LIN {X 0,Y 417.508,Z 538.945,A -85,B 0,C 180,E1 -10179.202,E2 -10179.202} C_VEL
LIN {X 0,Y 417.931,Z 531.783,A -85,B 0,C 180,E1 -10180.905,E2 -10180.905} C_VEL
LIN {X 0,Y 418.426,Z 524.272,A -85,B 0,C 180,E1 -10182.366,E2 -10182.366} C_VEL
LIN {X 0,Y 419.126,Z 515.227,A -85,B 0,C 180,E1 -10183.824,E2 -10183.824} C_VEL
LIN {X 0,Y 419.941,Z 504.249,A -85,B 0,C 180,E1 -10185.283,E2 -10185.283} C_VEL
LIN {X 0,Y 420.839,Z 493.102,A -85,B 0,C 180,E1 -10186.493,E2 -10186.493} C_VEL
LIN {X 0,Y 421.825,Z 480.792,A -85,B 0,C 180,E1 -10187.576,E2 -10187.576} C_VEL
LIN {X 0,Y 422.664,Z 467.695,A -85,B 0,C 180,E1 -10188.494,E2 -10188.494} C_VEL
LIN {X 0,Y 423.488,Z 453.313,A -85,B 0,C 180,E1 -10189.262,E2 -10189.262} C_VEL
LIN {X 0,Y 424.154,Z 439.428,A -85,B 0,C 180,E1 -10189.794,E2 -10189.794} C_VEL
LIN {X 0,Y 424.598,Z 424.854,A -85,B 0,C 180,E1 -10190.15,E2 -10190.15} C_VEL
LIN {X 0,Y 426.165,Z 318.753,A -85,B 0,C 180,E1 -10192.051,E2 -10192.051} C_VEL
LIN {X 0,Y 422.715,Z 297.962,A -85,B 0,C 180,E1 -10192.643,E2 -10192.643} C_VEL
LIN {X 0,Y 424.107,Z 281.691,A -85,B 0,C 180,E1 -10195.259,E2 -10195.259} C_VEL
LIN {X 0,Y 423.846,Z 278.694,A -85,B 0,C 180,E1 -10195.785,E2 -10195.785} C_VEL
LIN {X 0,Y 420.942,Z 266.303,A -85,B 0,C 180,E1 -10198.141,E2 -10198.141} C_VEL
LIN {X 0,Y 418.292,Z 256.11,A -85,B 0,C 180,E1 -10200.218,E2 -10200.218} C_VEL
LIN {X 0,Y 418.246,Z 256.011,A -85,B 0,C 180,E1 -10203.677,E2 -10203.677} C_VEL
LIN {X 0,Y 418.237,Z 255.991,A -85,B 0,C 180,E1 -10207.224,E2 -10207.224} C_VEL
LIN {X 0,Y 418.246,Z 256.012,A -85,B 0,C 180,E1 -10209.682,E2 -10209.682} C_VEL
LIN {X 0,Y 418.281,Z 256.01,A -85,B 0,C 180,E1 -10212.329,E2 -10212.329} C_VEL
LIN {X 0,Y 418.248,Z 256.006,A -85,B 0,C 180,E1 -10215.11,E2 -10215.11} C_VEL
LIN {X 0,Y 418.236,Z 256.008,A -85,B 0,C 180,E1 -10217.767,E2 -10217.767} C_VEL
LIN {X 0,Y 418.255,Z 256.011,A -85,B 0,C 180,E1 -10220.618,E2 -10220.618} C_VEL
LIN {X 0,Y 418.241,Z 255.998,A -85,B 0,C 180,E1 -10223.976,E2 -10223.976} C_VEL
LIN {X 0,Y 418.253,Z 256.009,A -85,B 0,C 180,E1 -10227.156,E2 -10227.156} C_VEL
LIN {X 0,Y 418.269,Z 255.993,A -85,B 0,C 180,E1 -10230.839,E2 -10230.839} C_VEL
LIN {X 0,Y 418.265,Z 256.01,A -85,B 0,C 180,E1 -10234.096,E2 -10234.096} C_VEL
LIN {X 0,Y 418.232,Z 256.011,A -85,B 0,C 180,E1 -10237.264,E2 -10237.264} C_VEL
LIN {X 0,Y 418.277,Z 256.006,A -85,B 0,C 180,E1 -10240.364,E2 -10240.364} C_VEL
LIN {X 0,Y 418.311,Z 256,A -85,B 0,C 180,E1 -10243.405,E2 -10243.405} C_VEL
LIN {X 0,Y 418.34,Z 255.996,A -85,B 0,C 180,E1 -10246.999,E2 -10246.999} C_VEL
LIN {X 0,Y 418.335,Z 255.998,A -85,B 0,C 180,E1 -10250.329,E2 -10250.329} C_VEL
LIN {X 0,Y 418.486,Z 255.973,A -85,B 0,C 180,E1 -10253.249,E2 -10253.249} C_VEL
LIN {X 0,Y 418.335,Z 256,A -85,B 0,C 180,E1 -10255.182,E2 -10255.182} C_VEL
LIN {X 0,Y 418.539,Z 255.971,A -85,B 0,C 180,E1 -10258.076,E2 -10258.076} C_VEL
LIN {X 0,Y 418.666,Z 255.958,A -85,B 0,C 180,E1 -10260,E2 -10260} C_VEL
LIN {X 0,Y 418.505,Z 255.971,A -85,B 0,C 180,E1 -10262.888,E2 -10262.888} C_VEL
LIN {X 0,Y 418.488,Z 255.974,A -85,B 0,C 180,E1 -10266.751,E2 -10266.751} C_VEL
LIN {X 0,Y 418.394,Z 255.989,A -85,B 0,C 180,E1 -10268.696,E2 -10268.696} C_VEL
LIN {X 0,Y 418.31,Z 255.998,A -85,B 0,C 180,E1 -10271.632,E2 -10271.632} C_VEL
LIN {X 0,Y 418.298,Z 256.002,A -85,B 0,C 180,E1 -10274.598,E2 -10274.598} C_VEL
LIN {X 0,Y 418.283,Z 256.007,A -85,B 0,C 180,E1 -10277.604,E2 -10277.604} C_VEL
LIN {X 0,Y 418.245,Z 256.005,A -85,B 0,C 180,E1 -10280.664,E2 -10280.664} C_VEL
LIN {X 0,Y 418.284,Z 256.002,A -85,B 0,C 180,E1 -10283.782,E2 -10283.782} C_VEL
LIN {X 0,Y 418.307,Z 255.999,A -85,B 0,C 180,E1 -10287.071,E2 -10287.071} C_VEL
LIN {X 0,Y 418.241,Z 256.001,A -85,B 0,C 180,E1 -10290.273,E2 -10290.273} C_VEL
LIN {X 0,Y 418.246,Z 256.004,A -85,B 0,C 180,E1 -10293.678,E2 -10293.678} C_VEL
LIN {X 0,Y 418.243,Z 256.014,A -85,B 0,C 180,E1 -10297.224,E2 -10297.224} C_VEL
LIN {X 0,Y 418.246,Z 255.998,A -85,B 0,C 180,E1 -10299.683,E2 -10299.683} C_VEL
LIN {X 0,Y 418.228,Z 256.014,A -85,B 0,C 180,E1 -10302.322,E2 -10302.322} C_VEL
LIN {X 0,Y 418.239,Z 256.011,A -85,B 0,C 180,E1 -10305.11,E2 -10305.11} C_VEL
LIN {X 0,Y 418.242,Z 256.004,A -85,B 0,C 180,E1 -10307.768,E2 -10307.768} C_VEL
LIN {X 0,Y 418.259,Z 255.993,A -85,B 0,C 180,E1 -10310.619,E2 -10310.619} C_VEL
LIN {X 0,Y 418.243,Z 256.013,A -85,B 0,C 180,E1 -10313.977,E2 -10313.977} C_VEL
LIN {X 0,Y 418.255,Z 256.107,A -85,B 0,C 180,E1 -10317.276,E2 -10317.276} C_VEL
LIN {X 0,Y 421.436,Z 269.127,A -85,B 0,C 180,E1 -10320.132,E2 -10320.132} C_VEL
LIN {X 0,Y 423.369,Z 278.645,A -85,B 0,C 180,E1 -10322.1,E2 -10322.1} C_VEL
LIN {X 0,Y 422.447,Z 290.987,A -85,B 0,C 180,E1 -10324.371,E2 -10324.371} C_VEL
LIN {X 0,Y 421.363,Z 305.324,A -85,B 0,C 180,E1 -10326.963,E2 -10326.963} C_VEL
LIN {X 0,Y 420.9,Z 313.173,A -85,B 0,C 180,E1 -10328.32,E2 -10328.32} C_VEL
LIN {X 0,Y 425.453,Z 338.255,A -85,B 0,C 180,E1 -10329.003,E2 -10329.003} C_VEL
LIN {X 0,Y 424.456,Z 426.611,A -85,B 0,C 180,E1 -10330.441,E2 -10330.441} C_VEL
LIN {X 0,Y 423.954,Z 439.651,A -85,B 0,C 180,E1 -10330.843,E2 -10330.843} C_VEL
LIN {X 0,Y 423.469,Z 452.234,A -85,B 0,C 180,E1 -10331.433,E2 -10331.433} C_VEL
LIN {X 0,Y 422.684,Z 464.51,A -85,B 0,C 180,E1 -10332.211,E2 -10332.211} C_VEL
LIN {X 0,Y 421.704,Z 476.092,A -85,B 0,C 180,E1 -10333.168,E2 -10333.168} C_VEL
LIN {X 0,Y 420.799,Z 486.5,A -85,B 0,C 180,E1 -10334.253,E2 -10334.253} C_VEL
LIN {X 0,Y 419.845,Z 496.326,A -85,B 0,C 180,E1 -10335.523,E2 -10335.523} C_VEL
LIN {X 0,Y 419.149,Z 503.803,A -85,B 0,C 180,E1 -10336.704,E2 -10336.704} C_VEL
LIN {X 0,Y 418.6,Z 511.176,A -85,B 0,C 180,E1 -10338.132,E2 -10338.132} C_VEL
LIN {X 0,Y 418.229,Z 514.558,A -85,B 0,C 180,E1 -10338.9,E2 -10338.9} C_VEL
LIN {X 0,Y 417.29,Z 517.409,A -85,B 0,C 180,E1 -10339.603,E2 -10339.603} C_VEL
LIN {X 0,Y 414.133,Z 521.613,A -85,B 0,C 180,E1 -10340.763,E2 -10340.763} C_VEL
LIN {X 0,Y 411.055,Z 525.123,A -85,B 0,C 180,E1 -10341.978,E2 -10341.978} C_VEL
LIN {X 0,Y 410.253,Z 526.877,A -85,B 0,C 180,E1 -10342.756,E2 -10342.756} C_VEL
LIN {X 0,Y 410.07,Z 529.255,A -85,B 0,C 180,E1 -10344.098,E2 -10344.098} C_VEL
LIN {X 0,Y 410.043,Z 530.517,A -85,B 0,C 180,E1 -10345.084,E2 -10345.084} C_VEL
LIN {X 0,Y 409.969,Z 531.939,A -85,B 0,C 180,E1 -10347.052,E2 -10347.052} C_VEL
LIN {X 0,Y 410.003,Z 532.078,A -85,B 0,C 180,E1 -10348.035,E2 -10348.035} C_VEL
LIN {X 0,Y 409.931,Z 531.25,A -85,B 0,C 180,E1 -10350,E2 -10350} C_VEL
LIN {X 0,Y 410.075,Z 528.965,A -85,B 0,C 180,E1 -10351.964,E2 -10351.964} C_VEL
LIN {X 0,Y 410.324,Z 526.18,A -85,B 0,C 180,E1 -10353.437,E2 -10353.437} C_VEL
LIN {X 0,Y 410.454,Z 522.443,A -85,B 0,C 180,E1 -10354.911,E2 -10354.911} C_VEL
LIN {X 0,Y 410.864,Z 517.636,A -85,B 0,C 180,E1 -10356.383,E2 -10356.383} C_VEL
LIN {X 0,Y 411.338,Z 511.624,A -85,B 0,C 180,E1 -10357.856,E2 -10357.856} C_VEL
LIN {X 0,Y 411.984,Z 504.185,A -85,B 0,C 180,E1 -10359.326,E2 -10359.326} C_VEL
LIN {X 0,Y 412.859,Z 494.877,A -85,B 0,C 180,E1 -10360.792,E2 -10360.792} C_VEL
LIN {X 0,Y 413.798,Z 484.254,A -85,B 0,C 180,E1 -10362.133,E2 -10362.133} C_VEL
LIN {X 0,Y 414.707,Z 473.337,A -85,B 0,C 180,E1 -10363.225,E2 -10363.225} C_VEL
LIN {X 0,Y 415.303,Z 464.403,A -85,B 0,C 180,E1 -10363.954,E2 -10363.954} C_VEL
LIN {X 0,Y 416.025,Z 453.249,A -85,B 0,C 180,E1 -10364.678,E2 -10364.678} C_VEL
LIN {X 0,Y 416.72,Z 440.712,A -85,B 0,C 180,E1 -10365.278,E2 -10365.278} C_VEL
LIN {X 0,Y 417.121,Z 427.911,A -85,B 0,C 180,E1 -10365.697,E2 -10365.697} C_VEL
LIN {X 0,Y 417.48,Z 404.6,A -85,B 0,C 180,E1 -10366.111,E2 -10366.111} C_VEL
LIN {X 0,Y 418.004,Z 337.982,A -85,B 0,C 180,E1 -10367.196,E2 -10367.196} C_VEL
LIN {X 0,Y 413.749,Z 313.265,A -85,B 0,C 180,E1 -10367.842,E2 -10367.842} C_VEL
LIN {X 0,Y 413.723,Z 312.244,A -85,B 0,C 180,E1 -10367.956,E2 -10367.956} C_VEL
LIN {X 0,Y 415.029,Z 293.533,A -85,B 0,C 180,E1 -10371.351,E2 -10371.351} C_VEL
LIN {X 0,Y 416.17,Z 279.659,A -85,B 0,C 180,E1 -10373.909,E2 -10373.909} C_VEL
LIN {X 0,Y 413.971,Z 268.598,A -85,B 0,C 180,E1 -10376.193,E2 -10376.193} C_VEL
LIN {X 0,Y 411.272,Z 256.972,A -85,B 0,C 180,E1 -10378.736,E2 -10378.736} C_VEL
LIN {X 0,Y 411.168,Z 256.892,A -85,B 0,C 180,E1 -10381.996,E2 -10381.996} C_VEL
LIN {X 0,Y 411.212,Z 256.877,A -85,B 0,C 180,E1 -10384.878,E2 -10384.878} C_VEL
LIN {X 0,Y 411.206,Z 256.884,A -85,B 0,C 180,E1 -10388.168,E2 -10388.168} C_VEL
LIN {X 0,Y 411.164,Z 256.887,A -85,B 0,C 180,E1 -10391.228,E2 -10391.228} C_VEL
LIN {X 0,Y 411.179,Z 256.886,A -85,B 0,C 180,E1 -10394.489,E2 -10394.489} C_VEL
LIN {X 0,Y 411.175,Z 256.889,A -85,B 0,C 180,E1 -10398.194,E2 -10398.194} C_VEL
LIN {X 0,Y 411.21,Z 256.873,A -85,B 0,C 180,E1 -10400.774,E2 -10400.774} C_VEL
LIN {X 0,Y 411.197,Z 256.887,A -85,B 0,C 180,E1 -10404.471,E2 -10404.471} C_VEL
LIN {X 0,Y 411.204,Z 256.87,A -85,B 0,C 180,E1 -10406.872,E2 -10406.872} C_VEL
LIN {X 0,Y 411.237,Z 256.886,A -85,B 0,C 180,E1 -10410.641,E2 -10410.641} C_VEL
LIN {X 0,Y 411.234,Z 256.883,A -85,B 0,C 180,E1 -10413.618,E2 -10413.618} C_VEL
LIN {X 0,Y 411.192,Z 256.888,A -85,B 0,C 180,E1 -10416.851,E2 -10416.851} C_VEL
LIN {X 0,Y 411.209,Z 256.881,A -85,B 0,C 180,E1 -10420.05,E2 -10420.05} C_VEL
LIN {X 0,Y 411.258,Z 256.88,A -85,B 0,C 180,E1 -10423.13,E2 -10423.13} C_VEL
LIN {X 0,Y 411.3,Z 256.879,A -85,B 0,C 180,E1 -10426.895,E2 -10426.895} C_VEL
LIN {X 0,Y 411.287,Z 256.871,A -85,B 0,C 180,E1 -10430.161,E2 -10430.161} C_VEL
LIN {X 0,Y 411.45,Z 256.856,A -85,B 0,C 180,E1 -10433.132,E2 -10433.132} C_VEL
LIN {X 0,Y 411.305,Z 256.866,A -85,B 0,C 180,E1 -10435.099,E2 -10435.099} C_VEL
LIN {X 0,Y 411.507,Z 256.85,A -85,B 0,C 180,E1 -10438.042,E2 -10438.042} C_VEL
LIN {X 0,Y 411.635,Z 256.831,A -85,B 0,C 180,E1 -10440,E2 -10440} C_VEL
LIN {X 0,Y 411.459,Z 256.856,A -85,B 0,C 180,E1 -10442.937,E2 -10442.937} C_VEL
LIN {X 0,Y 411.453,Z 256.854,A -85,B 0,C 180,E1 -10446.867,E2 -10446.867} C_VEL
LIN {X 0,Y 411.347,Z 256.869,A -85,B 0,C 180,E1 -10448.845,E2 -10448.845} C_VEL
LIN {X 0,Y 411.277,Z 256.872,A -85,B 0,C 180,E1 -10451.833,E2 -10451.833} C_VEL
LIN {X 0,Y 411.253,Z 256.877,A -85,B 0,C 180,E1 -10454.853,E2 -10454.853} C_VEL
LIN {X 0,Y 411.246,Z 256.883,A -85,B 0,C 180,E1 -10457.915,E2 -10457.915} C_VEL
LIN {X 0,Y 411.19,Z 256.884,A -85,B 0,C 180,E1 -10461.034,E2 -10461.034} C_VEL
LIN {X 0,Y 411.22,Z 256.883,A -85,B 0,C 180,E1 -10464.216,E2 -10464.216} C_VEL
LIN {X 0,Y 411.254,Z 256.882,A -85,B 0,C 180,E1 -10467.478,E2 -10467.478} C_VEL
LIN {X 0,Y 411.192,Z 256.872,A -85,B 0,C 180,E1 -10470.847,E2 -10470.847} C_VEL
LIN {X 0,Y 411.201,Z 256.888,A -85,B 0,C 180,E1 -10474.334,E2 -10474.334} C_VEL
LIN {X 0,Y 411.196,Z 256.881,A -85,B 0,C 180,E1 -10477.973,E2 -10477.973} C_VEL
LIN {X 0,Y 411.178,Z 256.889,A -85,B 0,C 180,E1 -10480.504,E2 -10480.504} C_VEL
LIN {X 0,Y 411.169,Z 256.886,A -85,B 0,C 180,E1 -10483.134,E2 -10483.134} C_VEL
LIN {X 0,Y 411.164,Z 256.883,A -85,B 0,C 180,E1 -10485.881,E2 -10485.881} C_VEL
LIN {X 0,Y 411.16,Z 256.86,A -85,B 0,C 180,E1 -10488.772,E2 -10488.772} C_VEL
LIN {X 0,Y 411.203,Z 256.888,A -85,B 0,C 180,E1 -10491.832,E2 -10491.832} C_VEL
LIN {X 0,Y 411.208,Z 256.871,A -85,B 0,C 180,E1 -10495.122,E2 -10495.122} C_VEL
LIN {X 0,Y 411.163,Z 256.876,A -85,B 0,C 180,E1 -10498.003,E2 -10498.003} C_VEL
LIN {X 0,Y 411.24,Z 257.068,A -85,B 0,C 180,E1 -10499.867,E2 -10499.867} C_VEL
LIN {X 0,Y 414.703,Z 270.774,A -85,B 0,C 180,E1 -10502.581,E2 -10502.581} C_VEL
LIN {X 0,Y 416.945,Z 281.265,A -85,B 0,C 180,E1 -10504.544,E2 -10504.544} C_VEL
LIN {X 0,Y 415.497,Z 297.774,A -85,B 0,C 180,E1 -10507.248,E2 -10507.248} C_VEL
LIN {X 0,Y 418.94,Z 319.913,A -85,B 0,C 180,E1 -10507.874,E2 -10507.874} C_VEL
LIN {X 0,Y 417.188,Z 430.973,A -85,B 0,C 180,E1 -10509.894,E2 -10509.894} C_VEL
LIN {X 0,Y 416.62,Z 445.021,A -85,B 0,C 180,E1 -10510.318,E2 -10510.318} C_VEL
LIN {X 0,Y 415.957,Z 458.882,A -85,B 0,C 180,E1 -10510.942,E2 -10510.942} C_VEL
LIN {X 0,Y 415.259,Z 471.531,A -85,B 0,C 180,E1 -10511.701,E2 -10511.701} C_VEL
LIN {X 0,Y 414.285,Z 484.97,A -85,B 0,C 180,E1 -10512.73,E2 -10512.73} C_VEL
LIN {X 0,Y 413.404,Z 496.539,A -85,B 0,C 180,E1 -10513.837,E2 -10513.837} C_VEL
LIN {X 0,Y 412.579,Z 506.143,A -85,B 0,C 180,E1 -10514.944,E2 -10514.944} C_VEL
LIN {X 0,Y 411.84,Z 516.768,A -85,B 0,C 180,E1 -10516.42,E2 -10516.42} C_VEL
LIN {X 0,Y 411.257,Z 525.627,A -85,B 0,C 180,E1 -10517.917,E2 -10517.917} C_VEL
LIN {X 0,Y 410.611,Z 533.98,A -85,B 0,C 180,E1 -10519.647,E2 -10519.647} C_VEL
LIN {X 0,Y 410.328,Z 539.839,A -85,B 0,C 180,E1 -10521.133,E2 -10521.133} C_VEL
LIN {X 0,Y 410.152,Z 544.584,A -85,B 0,C 180,E1 -10522.617,E2 -10522.617} C_VEL
LIN {X 0,Y 409.985,Z 548.373,A -85,B 0,C 180,E1 -10524.097,E2 -10524.097} C_VEL
LIN {X 0,Y 409.976,Z 550.404,A -85,B 0,C 180,E1 -10525.083,E2 -10525.083} C_VEL
LIN {X 0,Y 409.921,Z 553.34,A -85,B 0,C 180,E1 -10527.052,E2 -10527.052} C_VEL
LIN {X 0,Y 409.964,Z 554.267,A -85,B 0,C 180,E1 -10528.035,E2 -10528.035} C_VEL
LIN {X 0,Y 409.924,Z 555.055,A -85,B 0,C 180,E1 -10530,E2 -10530} C_VEL
LIN {X 0,Y 409.964,Z 554.426,A -85,B 0,C 180,E1 -10531.965,E2 -10531.965} C_VEL
LIN {X 0,Y 409.918,Z 552.354,A -85,B 0,C 180,E1 -10533.932,E2 -10533.932} C_VEL
LIN {X 0,Y 410.004,Z 548.817,A -85,B 0,C 180,E1 -10535.903,E2 -10535.903} C_VEL
LIN {X 0,Y 410.185,Z 543.719,A -85,B 0,C 180,E1 -10537.878,E2 -10537.878} C_VEL
LIN {X 0,Y 410.474,Z 538.77,A -85,B 0,C 180,E1 -10539.361,E2 -10539.361} C_VEL
LIN {X 0,Y 410.926,Z 531.608,A -85,B 0,C 180,E1 -10541.093,E2 -10541.093} C_VEL
LIN {X 0,Y 411.588,Z 522.719,A -85,B 0,C 180,E1 -10542.825,E2 -10542.825} C_VEL
LIN {X 0,Y 412.298,Z 513.396,A -85,B 0,C 180,E1 -10544.31,E2 -10544.31} C_VEL
LIN {X 0,Y 413.146,Z 503.071,A -85,B 0,C 180,E1 -10545.667,E2 -10545.667} C_VEL
LIN {X 0,Y 414.147,Z 491.652,A -85,B 0,C 180,E1 -10546.894,E2 -10546.894} C_VEL
LIN {X 0,Y 415.173,Z 478.997,A -85,B 0,C 180,E1 -10547.995,E2 -10547.995} C_VEL
LIN {X 0,Y 415.992,Z 466.908,A -85,B 0,C 180,E1 -10548.838,E2 -10548.838} C_VEL
LIN {X 0,Y 416.76,Z 453.384,A -85,B 0,C 180,E1 -10549.569,E2 -10549.569} C_VEL
LIN {X 0,Y 417.464,Z 439.087,A -85,B 0,C 180,E1 -10550.124,E2 -10550.124} C_VEL
LIN {X 0,Y 417.928,Z 424.273,A -85,B 0,C 180,E1 -10550.486,E2 -10550.486} C_VEL
LIN {X 0,Y 419.563,Z 319.793,A -85,B 0,C 180,E1 -10552.386,E2 -10552.386} C_VEL
LIN {X 0,Y 415.969,Z 297.92,A -85,B 0,C 180,E1 -10553.031,E2 -10553.031} C_VEL
LIN {X 0,Y 417.324,Z 283.314,A -85,B 0,C 180,E1 -10555.431,E2 -10555.431} C_VEL
LIN {X 0,Y 416.994,Z 280.233,A -85,B 0,C 180,E1 -10555.989,E2 -10555.989} C_VEL
LIN {X 0,Y 414.402,Z 269.167,A -85,B 0,C 180,E1 -10558.129,E2 -10558.129} C_VEL
LIN {X 0,Y 411.232,Z 256.989,A -85,B 0,C 180,E1 -10560.647,E2 -10560.647} C_VEL
LIN {X 0,Y 411.204,Z 256.889,A -85,B 0,C 180,E1 -10564.333,E2 -10564.333} C_VEL
LIN {X 0,Y 411.191,Z 256.879,A -85,B 0,C 180,E1 -10567.973,E2 -10567.973} C_VEL
LIN {X 0,Y 411.202,Z 256.883,A -85,B 0,C 180,E1 -10571.235,E2 -10571.235} C_VEL
LIN {X 0,Y 411.224,Z 256.877,A -85,B 0,C 180,E1 -10574.483,E2 -10574.483} C_VEL
LIN {X 0,Y 411.174,Z 256.882,A -85,B 0,C 180,E1 -10578.194,E2 -10578.194} C_VEL
LIN {X 0,Y 411.219,Z 256.887,A -85,B 0,C 180,E1 -10580.776,E2 -10580.776} C_VEL
LIN {X 0,Y 411.195,Z 256.876,A -85,B 0,C 180,E1 -10584.471,E2 -10584.471} C_VEL
LIN {X 0,Y 411.202,Z 256.887,A -85,B 0,C 180,E1 -10586.873,E2 -10586.873} C_VEL
LIN {X 0,Y 411.235,Z 256.866,A -85,B 0,C 180,E1 -10590.642,E2 -10590.642} C_VEL
LIN {X 0,Y 411.232,Z 256.885,A -85,B 0,C 180,E1 -10593.619,E2 -10593.619} C_VEL
LIN {X 0,Y 411.197,Z 256.887,A -85,B 0,C 180,E1 -10596.852,E2 -10596.852} C_VEL
LIN {X 0,Y 411.209,Z 256.885,A -85,B 0,C 180,E1 -10600.05,E2 -10600.05} C_VEL
LIN {X 0,Y 411.257,Z 256.878,A -85,B 0,C 180,E1 -10603.131,E2 -10603.131} C_VEL
LIN {X 0,Y 411.299,Z 256.873,A -85,B 0,C 180,E1 -10606.896,E2 -10606.896} C_VEL
LIN {X 0,Y 411.287,Z 256.877,A -85,B 0,C 180,E1 -10610.161,E2 -10610.161} C_VEL
LIN {X 0,Y 411.45,Z 256.849,A -85,B 0,C 180,E1 -10613.133,E2 -10613.133} C_VEL
LIN {X 0,Y 411.306,Z 256.875,A -85,B 0,C 180,E1 -10615.099,E2 -10615.099} C_VEL
LIN {X 0,Y 411.508,Z 256.847,A -85,B 0,C 180,E1 -10618.043,E2 -10618.043} C_VEL
LIN {X 0,Y 411.636,Z 256.834,A -85,B 0,C 180,E1 -10620,E2 -10620} C_VEL
LIN {X 0,Y 411.46,Z 256.848,A -85,B 0,C 180,E1 -10622.938,E2 -10622.938} C_VEL
LIN {X 0,Y 411.455,Z 256.851,A -85,B 0,C 180,E1 -10626.867,E2 -10626.867} C_VEL
LIN {X 0,Y 411.349,Z 256.868,A -85,B 0,C 180,E1 -10628.846,E2 -10628.846} C_VEL
LIN {X 0,Y 411.278,Z 256.875,A -85,B 0,C 180,E1 -10631.833,E2 -10631.833} C_VEL
LIN {X 0,Y 411.255,Z 256.881,A -85,B 0,C 180,E1 -10634.853,E2 -10634.853} C_VEL
LIN {X 0,Y 411.248,Z 256.881,A -85,B 0,C 180,E1 -10637.916,E2 -10637.916} C_VEL
LIN {X 0,Y 411.192,Z 256.887,A -85,B 0,C 180,E1 -10641.035,E2 -10641.035} C_VEL
LIN {X 0,Y 411.223,Z 256.88,A -85,B 0,C 180,E1 -10644.216,E2 -10644.216} C_VEL
LIN {X 0,Y 411.255,Z 256.872,A -85,B 0,C 180,E1 -10647.478,E2 -10647.478} C_VEL
LIN {X 0,Y 411.186,Z 256.884,A -85,B 0,C 180,E1 -10650.848,E2 -10650.848} C_VEL
LIN {X 0,Y 411.204,Z 256.879,A -85,B 0,C 180,E1 -10654.334,E2 -10654.334} C_VEL
LIN {X 0,Y 411.196,Z 256.888,A -85,B 0,C 180,E1 -10657.974,E2 -10657.974} C_VEL
LIN {X 0,Y 411.162,Z 256.891,A -85,B 0,C 180,E1 -10661.229,E2 -10661.229} C_VEL
LIN {X 0,Y 411.176,Z 256.883,A -85,B 0,C 180,E1 -10664.491,E2 -10664.491} C_VEL
LIN {X 0,Y 411.179,Z 256.885,A -85,B 0,C 180,E1 -10668.196,E2 -10668.196} C_VEL
LIN {X 0,Y 411.223,Z 256.866,A -85,B 0,C 180,E1 -10670.777,E2 -10670.777} C_VEL
LIN {X 0,Y 411.198,Z 256.887,A -85,B 0,C 180,E1 -10674.472,E2 -10674.472} C_VEL
LIN {X 0,Y 411.246,Z 257.106,A -85,B 0,C 180,E1 -10676.907,E2 -10676.907} C_VEL
LIN {X 0,Y 414.73,Z 271.34,A -85,B 0,C 180,E1 -10680.067,E2 -10680.067} C_VEL
LIN {X 0,Y 416.458,Z 279.57,A -85,B 0,C 180,E1 -10681.803,E2 -10681.803} C_VEL
LIN {X 0,Y 416.228,Z 285.218,A -85,B 0,C 180,E1 -10682.878,E2 -10682.878} C_VEL
LIN {X 0,Y 414.746,Z 303.298,A -85,B 0,C 180,E1 -10686.214,E2 -10686.214} C_VEL
LIN {X 0,Y 414.075,Z 312.742,A -85,B 0,C 180,E1 -10687.911,E2 -10687.911} C_VEL
LIN {X 0,Y 415.375,Z 319.839,A -85,B 0,C 180,E1 -10688.147,E2 -10688.147} C_VEL
LIN {X 0,Y 418.719,Z 338.165,A -85,B 0,C 180,E1 -10688.644,E2 -10688.644} C_VEL
LIN {X 0,Y 417.779,Z 426.746,A -85,B 0,C 180,E1 -10690.116,E2 -10690.116} C_VEL
LIN {X 0,Y 417.246,Z 440.288,A -85,B 0,C 180,E1 -10690.544,E2 -10690.544} C_VEL
LIN {X 0,Y 416.72,Z 452.62,A -85,B 0,C 180,E1 -10691.136,E2 -10691.136} C_VEL
LIN {X 0,Y 415.918,Z 464.616,A -85,B 0,C 180,E1 -10691.911,E2 -10691.911} C_VEL
LIN {X 0,Y 414.908,Z 476.201,A -85,B 0,C 180,E1 -10692.884,E2 -10692.884} C_VEL
LIN {X 0,Y 413.939,Z 486.615,A -85,B 0,C 180,E1 -10693.985,E2 -10693.985} C_VEL
LIN {X 0,Y 412.989,Z 496.018,A -85,B 0,C 180,E1 -10695.211,E2 -10695.211} C_VEL
LIN {X 0,Y 412.156,Z 504.452,A -85,B 0,C 180,E1 -10696.57,E2 -10696.57} C_VEL
LIN {X 0,Y 411.628,Z 511.313,A -85,B 0,C 180,E1 -10697.927,E2 -10697.927} C_VEL
LIN {X 0,Y 411.024,Z 516.496,A -85,B 0,C 180,E1 -10699.159,E2 -10699.159} C_VEL
LIN {X 0,Y 410.606,Z 521.559,A -85,B 0,C 180,E1 -10700.642,E2 -10700.642} C_VEL
LIN {X 0,Y 410.356,Z 525.512,A -85,B 0,C 180,E1 -10702.125,E2 -10702.125} C_VEL
LIN {X 0,Y 410.253,Z 526.877,A -85,B 0,C 180,E1 -10702.756,E2 -10702.756} C_VEL
LIN {X 0,Y 409.461,Z 528.427,A -85,B 0,C 180,E1 -10703.546,E2 -10703.546} C_VEL
LIN {X 0,Y 406.473,Z 530.506,A -85,B 0,C 180,E1 -10704.843,E2 -10704.843} C_VEL
LIN {X 0,Y 404.009,Z 531.615,A -85,B 0,C 180,E1 -10705.904,E2 -10705.904} C_VEL
LIN {X 0,Y 402.955,Z 532.065,A -85,B 0,C 180,E1 -10706.73,E2 -10706.73} C_VEL
LIN {X 0,Y 402.869,Z 532.13,A -85,B 0,C 180,E1 -10707.011,E2 -10707.011} C_VEL
LIN {X 0,Y 402.915,Z 532.28,A -85,B 0,C 180,E1 -10708.001,E2 -10708.001} C_VEL
LIN {X 0,Y 402.855,Z 531.466,A -85,B 0,C 180,E1 -10710,E2 -10710} C_VEL
LIN {X 0,Y 403.008,Z 529.197,A -85,B 0,C 180,E1 -10711.999,E2 -10711.999} C_VEL
LIN {X 0,Y 403.264,Z 526.429,A -85,B 0,C 180,E1 -10713.497,E2 -10713.497} C_VEL
LIN {X 0,Y 403.391,Z 522.713,A -85,B 0,C 180,E1 -10714.997,E2 -10714.997} C_VEL
LIN {X 0,Y 403.832,Z 517.928,A -85,B 0,C 180,E1 -10716.495,E2 -10716.495} C_VEL
LIN {X 0,Y 404.447,Z 510.835,A -85,B 0,C 180,E1 -10718.242,E2 -10718.242} C_VEL
LIN {X 0,Y 405.151,Z 503.117,A -85,B 0,C 180,E1 -10719.737,E2 -10719.737} C_VEL
LIN {X 0,Y 406.079,Z 493.542,A -85,B 0,C 180,E1 -10721.227,E2 -10721.227} C_VEL
LIN {X 0,Y 406.959,Z 483.66,A -85,B 0,C 180,E1 -10722.466,E2 -10722.466} C_VEL
LIN {X 0,Y 407.94,Z 472.506,A -85,B 0,C 180,E1 -10723.576,E2 -10723.576} C_VEL
LIN {X 0,Y 408.617,Z 463.379,A -85,B 0,C 180,E1 -10724.314,E2 -10724.314} C_VEL
LIN {X 0,Y 409.399,Z 450.726,A -85,B 0,C 180,E1 -10725.112,E2 -10725.112} C_VEL
LIN {X 0,Y 410.068,Z 438.01,A -85,B 0,C 180,E1 -10725.692,E2 -10725.692} C_VEL
LIN {X 0,Y 410.468,Z 424.986,A -85,B 0,C 180,E1 -10726.08,E2 -10726.08} C_VEL
LIN {X 0,Y 411.371,Z 339.141,A -85,B 0,C 180,E1 -10727.509,E2 -10727.509} C_VEL
LIN {X 0,Y 406.871,Z 312.737,A -85,B 0,C 180,E1 -10728.229,E2 -10728.229} C_VEL
LIN {X 0,Y 408.189,Z 294.301,A -85,B 0,C 180,E1 -10731.603,E2 -10731.603} C_VEL
LIN {X 0,Y 409.328,Z 281.156,A -85,B 0,C 180,E1 -10734.065,E2 -10734.065} C_VEL
LIN {X 0,Y 406.796,Z 268.704,A -85,B 0,C 180,E1 -10736.691,E2 -10736.691} C_VEL
LIN {X 0,Y 404.213,Z 257.842,A -85,B 0,C 180,E1 -10739.132,E2 -10739.132} C_VEL
LIN {X 0,Y 404.143,Z 257.754,A -85,B 0,C 180,E1 -10742.621,E2 -10742.621} C_VEL
LIN {X 0,Y 404.182,Z 257.755,A -85,B 0,C 180,E1 -10745.189,E2 -10745.189} C_VEL
LIN {X 0,Y 404.156,Z 257.764,A -85,B 0,C 180,E1 -10748.756,E2 -10748.756} C_VEL
LIN {X 0,Y 404.124,Z 257.765,A -85,B 0,C 180,E1 -10751.599,E2 -10751.599} C_VEL
LIN {X 0,Y 404.148,Z 257.761,A -85,B 0,C 180,E1 -10754.522,E2 -10754.522} C_VEL
LIN {X 0,Y 404.135,Z 257.772,A -85,B 0,C 180,E1 -10757.295,E2 -10757.295} C_VEL
LIN {X 0,Y 404.167,Z 257.747,A -85,B 0,C 180,E1 -10759.954,E2 -10759.954} C_VEL
LIN {X 0,Y 404.137,Z 257.772,A -85,B 0,C 180,E1 -10763.124,E2 -10763.124} C_VEL
LIN {X 0,Y 404.142,Z 257.747,A -85,B 0,C 180,E1 -10766.187,E2 -10766.187} C_VEL
LIN {X 0,Y 404.151,Z 257.766,A -85,B 0,C 180,E1 -10769.715,E2 -10769.715} C_VEL
LIN {X 0,Y 404.192,Z 257.764,A -85,B 0,C 180,E1 -10773.122,E2 -10773.122} C_VEL
LIN {X 0,Y 404.17,Z 257.757,A -85,B 0,C 180,E1 -10775.333,E2 -10775.333} C_VEL
LIN {X 0,Y 404.154,Z 257.769,A -85,B 0,C 180,E1 -10778.581,E2 -10778.581} C_VEL
LIN {X 0,Y 404.205,Z 257.757,A -85,B 0,C 180,E1 -10781.761,E2 -10781.761} C_VEL
LIN {X 0,Y 404.202,Z 257.754,A -85,B 0,C 180,E1 -10784.881,E2 -10784.881} C_VEL
LIN {X 0,Y 404.251,Z 257.753,A -85,B 0,C 180,E1 -10787.958,E2 -10787.958} C_VEL
LIN {X 0,Y 404.399,Z 257.734,A -85,B 0,C 180,E1 -10792.128,E2 -10792.128} C_VEL
LIN {X 0,Y 404.416,Z 257.732,A -85,B 0,C 180,E1 -10794.015,E2 -10794.015} C_VEL
LIN {X 0,Y 404.476,Z 257.726,A -85,B 0,C 180,E1 -10798.008,E2 -10798.008} C_VEL
LIN {X 0,Y 404.604,Z 257.707,A -85,B 0,C 180,E1 -10800,E2 -10800} C_VEL
LIN {X 0,Y 404.417,Z 257.733,A -85,B 0,C 180,E1 -10802.988,E2 -10802.988} C_VEL
LIN {X 0,Y 404.405,Z 257.731,A -85,B 0,C 180,E1 -10806.987,E2 -10806.987} C_VEL
LIN {X 0,Y 404.251,Z 257.753,A -85,B 0,C 180,E1 -10810.012,E2 -10810.012} C_VEL
LIN {X 0,Y 404.26,Z 257.751,A -85,B 0,C 180,E1 -10813.211,E2 -10813.211} C_VEL
LIN {X 0,Y 404.209,Z 257.756,A -85,B 0,C 180,E1 -10817.007,E2 -10817.007} C_VEL
LIN {X 0,Y 404.157,Z 257.761,A -85,B 0,C 180,E1 -10820.352,E2 -10820.352} C_VEL
LIN {X 0,Y 404.163,Z 257.765,A -85,B 0,C 180,E1 -10823.575,E2 -10823.575} C_VEL
LIN {X 0,Y 404.177,Z 257.76,A -85,B 0,C 180,E1 -10825.767,E2 -10825.767} C_VEL
LIN {X 0,Y 404.192,Z 257.759,A -85,B 0,C 180,E1 -10828,E2 -10828} C_VEL
LIN {X 0,Y 404.137,Z 257.754,A -85,B 0,C 180,E1 -10831.559,E2 -10831.559} C_VEL
LIN {X 0,Y 404.18,Z 257.76,A -85,B 0,C 180,E1 -10835.016,E2 -10835.016} C_VEL
LIN {X 0,Y 404.154,Z 257.765,A -85,B 0,C 180,E1 -10838.757,E2 -10838.757} C_VEL
LIN {X 0,Y 404.118,Z 257.763,A -85,B 0,C 180,E1 -10841.6,E2 -10841.6} C_VEL
LIN {X 0,Y 404.142,Z 257.767,A -85,B 0,C 180,E1 -10844.523,E2 -10844.523} C_VEL
LIN {X 0,Y 404.132,Z 257.737,A -85,B 0,C 180,E1 -10847.296,E2 -10847.296} C_VEL
LIN {X 0,Y 404.165,Z 257.748,A -85,B 0,C 180,E1 -10849.956,E2 -10849.956} C_VEL
LIN {X 0,Y 404.133,Z 257.752,A -85,B 0,C 180,E1 -10853.126,E2 -10853.126} C_VEL
LIN {X 0,Y 404.142,Z 257.771,A -85,B 0,C 180,E1 -10856.188,E2 -10856.188} C_VEL
LIN {X 0,Y 404.189,Z 257.957,A -85,B 0,C 180,E1 -10859.467,E2 -10859.467} C_VEL
LIN {X 0,Y 407.319,Z 270.219,A -85,B 0,C 180,E1 -10861.958,E2 -10861.958} C_VEL
LIN {X 0,Y 410.071,Z 282.717,A -85,B 0,C 180,E1 -10864.359,E2 -10864.359} C_VEL
LIN {X 0,Y 408.835,Z 296.689,A -85,B 0,C 180,E1 -10866.711,E2 -10866.711} C_VEL
LIN {X 0,Y 408.735,Z 298.114,A -85,B 0,C 180,E1 -10866.912,E2 -10866.912} C_VEL
LIN {X 0,Y 412.249,Z 320.698,A -85,B 0,C 180,E1 -10867.55,E2 -10867.55} C_VEL
LIN {X 0,Y 410.441,Z 430.67,A -85,B 0,C 180,E1 -10869.581,E2 -10869.581} C_VEL
LIN {X 0,Y 409.876,Z 444.755,A -85,B 0,C 180,E1 -10870.01,E2 -10870.01} C_VEL
LIN {X 0,Y 409.183,Z 458.401,A -85,B 0,C 180,E1 -10870.628,E2 -10870.628} C_VEL
LIN {X 0,Y 408.434,Z 471.698,A -85,B 0,C 180,E1 -10871.44,E2 -10871.44} C_VEL
LIN {X 0,Y 407.481,Z 484.467,A -85,B 0,C 180,E1 -10872.433,E2 -10872.433} C_VEL
LIN {X 0,Y 406.503,Z 496.097,A -85,B 0,C 180,E1 -10873.555,E2 -10873.555} C_VEL
LIN {X 0,Y 405.64,Z 505.752,A -85,B 0,C 180,E1 -10874.68,E2 -10874.68} C_VEL
LIN {X 0,Y 404.88,Z 516.255,A -85,B 0,C 180,E1 -10876.157,E2 -10876.157} C_VEL
LIN {X 0,Y 404.234,Z 525.307,A -85,B 0,C 180,E1 -10877.703,E2 -10877.703} C_VEL
LIN {X 0,Y 403.592,Z 533.699,A -85,B 0,C 180,E1 -10879.465,E2 -10879.465} C_VEL
LIN {X 0,Y 403.274,Z 539.571,A -85,B 0,C 180,E1 -10880.976,E2 -10880.976} C_VEL
LIN {X 0,Y 403.059,Z 544.331,A -85,B 0,C 180,E1 -10882.486,E2 -10882.486} C_VEL
LIN {X 0,Y 402.917,Z 548.138,A -85,B 0,C 180,E1 -10883.993,E2 -10883.993} C_VEL
LIN {X 0,Y 402.837,Z 551.832,A -85,B 0,C 180,E1 -10885.998,E2 -10885.998} C_VEL
LIN {X 0,Y 402.862,Z 554.055,A -85,B 0,C 180,E1 -10888.001,E2 -10888.001} C_VEL
LIN {X 0,Y 402.849,Z 554.854,A -85,B 0,C 180,E1 -10890,E2 -10890} C_VEL
LIN {X 0,Y 402.862,Z 554.234,A -85,B 0,C 180,E1 -10891.999,E2 -10891.999} C_VEL
LIN {X 0,Y 402.837,Z 552.17,A -85,B 0,C 180,E1 -10894.002,E2 -10894.002} C_VEL
LIN {X 0,Y 402.937,Z 548.638,A -85,B 0,C 180,E1 -10896.007,E2 -10896.007} C_VEL
LIN {X 0,Y 403.13,Z 543.543,A -85,B 0,C 180,E1 -10898.017,E2 -10898.017} C_VEL
LIN {X 0,Y 403.424,Z 538.596,A -85,B 0,C 180,E1 -10899.526,E2 -10899.526} C_VEL
LIN {X 0,Y 403.931,Z 531.437,A -85,B 0,C 180,E1 -10901.288,E2 -10901.288} C_VEL
LIN {X 0,Y 404.634,Z 522.547,A -85,B 0,C 180,E1 -10903.049,E2 -10903.049} C_VEL
LIN {X 0,Y 405.376,Z 513.223,A -85,B 0,C 180,E1 -10904.559,E2 -10904.559} C_VEL
LIN {X 0,Y 406.283,Z 502.894,A -85,B 0,C 180,E1 -10905.939,E2 -10905.939} C_VEL
LIN {X 0,Y 407.297,Z 491.465,A -85,B 0,C 180,E1 -10907.187,E2 -10907.187} C_VEL
LIN {X 0,Y 408.396,Z 478.965,A -85,B 0,C 180,E1 -10908.29,E2 -10908.29} C_VEL
LIN {X 0,Y 409.291,Z 466.146,A -85,B 0,C 180,E1 -10909.194,E2 -10909.194} C_VEL
LIN {X 0,Y 410.082,Z 453.126,A -85,B 0,C 180,E1 -10909.901,E2 -10909.901} C_VEL
LIN {X 0,Y 410.775,Z 438.759,A -85,B 0,C 180,E1 -10910.467,E2 -10910.467} C_VEL
LIN {X 0,Y 411.285,Z 423.714,A -85,B 0,C 180,E1 -10910.832,E2 -10910.832} C_VEL
LIN {X 0,Y 412.98,Z 320.585,A -85,B 0,C 180,E1 -10912.736,E2 -10912.736} C_VEL
LIN {X 0,Y 409.252,Z 298.303,A -85,B 0,C 180,E1 -10913.4,E2 -10913.4} C_VEL
LIN {X 0,Y 409.987,Z 290.296,A -85,B 0,C 180,E1 -10914.698,E2 -10914.698} C_VEL
LIN {X 0,Y 410.517,Z 284.914,A -85,B 0,C 180,E1 -10915.612,E2 -10915.612} C_VEL
LIN {X 0,Y 409.469,Z 278.612,A -85,B 0,C 180,E1 -10916.809,E2 -10916.809} C_VEL
LIN {X 0,Y 405.914,Z 264.367,A -85,B 0,C 180,E1 -10919.686,E2 -10919.686} C_VEL
LIN {X 0,Y 404.166,Z 257.844,A -85,B 0,C 180,E1 -10921.116,E2 -10921.116} C_VEL
LIN {X 0,Y 404.143,Z 257.769,A -85,B 0,C 180,E1 -10923.812,E2 -10923.812} C_VEL
LIN {X 0,Y 404.133,Z 257.742,A -85,B 0,C 180,E1 -10926.874,E2 -10926.874} C_VEL
LIN {X 0,Y 404.152,Z 257.764,A -85,B 0,C 180,E1 -10930.081,E2 -10930.081} C_VEL
LIN {X 0,Y 404.201,Z 257.759,A -85,B 0,C 180,E1 -10933.091,E2 -10933.091} C_VEL
LIN {X 0,Y 404.149,Z 257.765,A -85,B 0,C 180,E1 -10935.926,E2 -10935.926} C_VEL
LIN {X 0,Y 404.114,Z 257.758,A -85,B 0,C 180,E1 -10938.635,E2 -10938.635} C_VEL
LIN {X 0,Y 404.154,Z 257.766,A -85,B 0,C 180,E1 -10941.491,E2 -10941.491} C_VEL
LIN {X 0,Y 404.181,Z 257.754,A -85,B 0,C 180,E1 -10944.984,E2 -10944.984} C_VEL
LIN {X 0,Y 404.141,Z 257.759,A -85,B 0,C 180,E1 -10948.554,E2 -10948.554} C_VEL
LIN {X 0,Y 404.192,Z 257.753,A -85,B 0,C 180,E1 -10952,E2 -10952} C_VEL
LIN {X 0,Y 404.172,Z 257.761,A -85,B 0,C 180,E1 -10955.334,E2 -10955.334} C_VEL
LIN {X 0,Y 404.133,Z 257.764,A -85,B 0,C 180,E1 -10958.581,E2 -10958.581} C_VEL
LIN {X 0,Y 404.204,Z 257.763,A -85,B 0,C 180,E1 -10961.762,E2 -10961.762} C_VEL
LIN {X 0,Y 404.2,Z 257.756,A -85,B 0,C 180,E1 -10964.882,E2 -10964.882} C_VEL
LIN {X 0,Y 404.25,Z 257.748,A -85,B 0,C 180,E1 -10967.959,E2 -10967.959} C_VEL
LIN {X 0,Y 404.399,Z 257.727,A -85,B 0,C 180,E1 -10972.129,E2 -10972.129} C_VEL
LIN {X 0,Y 404.417,Z 257.734,A -85,B 0,C 180,E1 -10974.015,E2 -10974.015} C_VEL
LIN {X 0,Y 404.477,Z 257.722,A -85,B 0,C 180,E1 -10978.009,E2 -10978.009} C_VEL
LIN {X 0,Y 404.605,Z 257.71,A -85,B 0,C 180,E1 -10980,E2 -10980} C_VEL
LIN {X 0,Y 404.418,Z 257.726,A -85,B 0,C 180,E1 -10982.989,E2 -10982.989} C_VEL
LIN {X 0,Y 404.406,Z 257.728,A -85,B 0,C 180,E1 -10986.988,E2 -10986.988} C_VEL
LIN {X 0,Y 404.253,Z 257.751,A -85,B 0,C 180,E1 -10990.012,E2 -10990.012} C_VEL
LIN {X 0,Y 404.261,Z 257.753,A -85,B 0,C 180,E1 -10993.212,E2 -10993.212} C_VEL
LIN {X 0,Y 404.211,Z 257.756,A -85,B 0,C 180,E1 -10997.008,E2 -10997.008} C_VEL
LIN {X 0,Y 404.159,Z 257.758,A -85,B 0,C 180,E1 -11000.352,E2 -11000.352} C_VEL
LIN {X 0,Y 404.165,Z 257.76,A -85,B 0,C 180,E1 -11003.575,E2 -11003.575} C_VEL
LIN {X 0,Y 404.18,Z 257.763,A -85,B 0,C 180,E1 -11005.767,E2 -11005.767} C_VEL
LIN {X 0,Y 404.192,Z 257.749,A -85,B 0,C 180,E1 -11008,E2 -11008} C_VEL
LIN {X 0,Y 404.137,Z 257.77,A -85,B 0,C 180,E1 -11011.559,E2 -11011.559} C_VEL
LIN {X 0,Y 404.183,Z 257.749,A -85,B 0,C 180,E1 -11015.017,E2 -11015.017} C_VEL
LIN {X 0,Y 404.153,Z 257.762,A -85,B 0,C 180,E1 -11018.758,E2 -11018.758} C_VEL
LIN {X 0,Y 404.122,Z 257.77,A -85,B 0,C 180,E1 -11021.601,E2 -11021.601} C_VEL
LIN {X 0,Y 404.146,Z 257.759,A -85,B 0,C 180,E1 -11024.523,E2 -11024.523} C_VEL
LIN {X 0,Y 404.14,Z 257.761,A -85,B 0,C 180,E1 -11027.297,E2 -11027.297} C_VEL
LIN {X 0,Y 404.169,Z 257.761,A -85,B 0,C 180,E1 -11029.956,E2 -11029.956} C_VEL
LIN {X 0,Y 404.137,Z 257.754,A -85,B 0,C 180,E1 -11033.126,E2 -11033.126} C_VEL
LIN {X 0,Y 404.169,Z 257.81,A -85,B 0,C 180,E1 -11036.372,E2 -11036.372} C_VEL
LIN {X 0,Y 404.653,Z 259.745,A -85,B 0,C 180,E1 -11036.892,E2 -11036.892} C_VEL
LIN {X 0,Y 408.057,Z 273.729,A -85,B 0,C 180,E1 -11040.036,E2 -11040.036} C_VEL
LIN {X 0,Y 409.742,Z 282.261,A -85,B 0,C 180,E1 -11041.857,E2 -11041.857} C_VEL
LIN {X 0,Y 408.623,Z 294.98,A -85,B 0,C 180,E1 -11044.261,E2 -11044.261} C_VEL
LIN {X 0,Y 407.459,Z 309.114,A -85,B 0,C 180,E1 -11046.896,E2 -11046.896} C_VEL
LIN {X 0,Y 407.271,Z 312.947,A -85,B 0,C 180,E1 -11047.547,E2 -11047.547} C_VEL
LIN {X 0,Y 412.16,Z 339.354,A -85,B 0,C 180,E1 -11048.304,E2 -11048.304} C_VEL
LIN {X 0,Y 411.144,Z 425.671,A -85,B 0,C 180,E1 -11049.748,E2 -11049.748} C_VEL
LIN {X 0,Y 410.633,Z 438.676,A -85,B 0,C 180,E1 -11050.146,E2 -11050.146} C_VEL
LIN {X 0,Y 410.067,Z 451.984,A -85,B 0,C 180,E1 -11050.776,E2 -11050.776} C_VEL
LIN {X 0,Y 409.268,Z 463.02,A -85,B 0,C 180,E1 -11051.477,E2 -11051.477} C_VEL
LIN {X 0,Y 408.391,Z 473.693,A -85,B 0,C 180,E1 -11052.344,E2 -11052.344} C_VEL
LIN {X 0,Y 407.291,Z 484.612,A -85,B 0,C 180,E1 -11053.458,E2 -11053.458} C_VEL
LIN {X 0,Y 406.303,Z 494.38,A -85,B 0,C 180,E1 -11054.705,E2 -11054.705} C_VEL
LIN {X 0,Y 405.329,Z 503.626,A -85,B 0,C 180,E1 -11056.166,E2 -11056.166} C_VEL
LIN {X 0,Y 404.643,Z 511.45,A -85,B 0,C 180,E1 -11057.716,E2 -11057.716} C_VEL
LIN {X 0,Y 403.873,Z 518.438,A -85,B 0,C 180,E1 -11059.472,E2 -11059.472} C_VEL
LIN {X 0,Y 403.472,Z 523.128,A -85,B 0,C 180,E1 -11060.981,E2 -11060.981} C_VEL
LIN {X 0,Y 403.171,Z 527.23,A -85,B 0,C 180,E1 -11062.722,E2 -11062.722} C_VEL
LIN {X 0,Y 402.99,Z 529.428,A -85,B 0,C 180,E1 -11063.994,E2 -11063.994} C_VEL
LIN {X 0,Y 402.954,Z 530.696,A -85,B 0,C 180,E1 -11064.997,E2 -11064.997} C_VEL
LIN {X 0,Y 402.869,Z 532.13,A -85,B 0,C 180,E1 -11067.011,E2 -11067.011} C_VEL
LIN {X 0,Y 402.189,Z 532.302,A -85,B 0,C 180,E1 -11067.846,E2 -11067.846} C_VEL
LIN {X 0,Y 399.303,Z 532.06,A -85,B 0,C 180,E1 -11069.204,E2 -11069.204} C_VEL
LIN {X 0,Y 396.899,Z 531.423,A -85,B 0,C 180,E1 -11070.295,E2 -11070.295} C_VEL
LIN {X 0,Y 395.912,Z 530.613,A -85,B 0,C 180,E1 -11071.134,E2 -11071.134} C_VEL
LIN {X 0,Y 395.857,Z 530.225,A -85,B 0,C 180,E1 -11071.416,E2 -11071.416} C_VEL
LIN {X 0,Y 396.092,Z 527.707,A -85,B 0,C 180,E1 -11073.051,E2 -11073.051} C_VEL
LIN {X 0,Y 396.283,Z 524.35,A -85,B 0,C 180,E1 -11074.577,E2 -11074.577} C_VEL
LIN {X 0,Y 396.637,Z 519.957,A -85,B 0,C 180,E1 -11076.103,E2 -11076.103} C_VEL
LIN {X 0,Y 397.216,Z 513.283,A -85,B 0,C 180,E1 -11077.897,E2 -11077.897} C_VEL
LIN {X 0,Y 397.885,Z 506.211,A -85,B 0,C 180,E1 -11079.403,E2 -11079.403} C_VEL
LIN {X 0,Y 398.804,Z 497.382,A -85,B 0,C 180,E1 -11080.92,E2 -11080.92} C_VEL
LIN {X 0,Y 399.726,Z 488.324,A -85,B 0,C 180,E1 -11082.18,E2 -11082.18} C_VEL
LIN {X 0,Y 400.577,Z 478.304,A -85,B 0,C 180,E1 -11083.313,E2 -11083.313} C_VEL
LIN {X 0,Y 401.474,Z 467.228,A -85,B 0,C 180,E1 -11084.315,E2 -11084.315} C_VEL
LIN {X 0,Y 402.314,Z 456.785,A -85,B 0,C 180,E1 -11085.061,E2 -11085.061} C_VEL
LIN {X 0,Y 403.051,Z 444.251,A -85,B 0,C 180,E1 -11085.745,E2 -11085.745} C_VEL
LIN {X 0,Y 403.578,Z 431.16,A -85,B 0,C 180,E1 -11086.242,E2 -11086.242} C_VEL
LIN {X 0,Y 403.879,Z 417.062,A -85,B 0,C 180,E1 -11086.549,E2 -11086.549} C_VEL
LIN {X 0,Y 404.737,Z 340.147,A -85,B 0,C 180,E1 -11087.835,E2 -11087.835} C_VEL
LIN {X 0,Y 400.059,Z 312.99,A -85,B 0,C 180,E1 -11088.579,E2 -11088.579} C_VEL
LIN {X 0,Y 400.052,Z 311.948,A -85,B 0,C 180,E1 -11088.698,E2 -11088.698} C_VEL
LIN {X 0,Y 401.606,Z 292.378,A -85,B 0,C 180,E1 -11092.371,E2 -11092.371} C_VEL
LIN {X 0,Y 402.447,Z 282.964,A -85,B 0,C 180,E1 -11094.166,E2 -11094.166} C_VEL
LIN {X 0,Y 400.569,Z 273.261,A -85,B 0,C 180,E1 -11096.234,E2 -11096.234} C_VEL
LIN {X 0,Y 397.605,Z 260.501,A -85,B 0,C 180,E1 -11099.083,E2 -11099.083} C_VEL
LIN {X 0,Y 397.148,Z 258.702,A -85,B 0,C 180,E1 -11099.556,E2 -11099.556} C_VEL
LIN {X 0,Y 397.116,Z 258.621,A -85,B 0,C 180,E1 -11103.272,E2 -11103.272} C_VEL
LIN {X 0,Y 397.109,Z 258.645,A -85,B 0,C 180,E1 -11105.734,E2 -11105.734} C_VEL
LIN {X 0,Y 397.114,Z 258.644,A -85,B 0,C 180,E1 -11109.576,E2 -11109.576} C_VEL
LIN {X 0,Y 397.104,Z 258.644,A -85,B 0,C 180,E1 -11113.478,E2 -11113.478} C_VEL
LIN {X 0,Y 397.101,Z 258.64,A -85,B 0,C 180,E1 -11116.52,E2 -11116.52} C_VEL
LIN {X 0,Y 397.111,Z 258.626,A -85,B 0,C 180,E1 -11120.422,E2 -11120.422} C_VEL
LIN {X 0,Y 397.106,Z 258.641,A -85,B 0,C 180,E1 -11124.265,E2 -11124.265} C_VEL
LIN {X 0,Y 397.111,Z 258.623,A -85,B 0,C 180,E1 -11126.726,E2 -11126.726} C_VEL
LIN {X 0,Y 397.13,Z 258.641,A -85,B 0,C 180,E1 -11130.296,E2 -11130.296} C_VEL
LIN {X 0,Y 397.191,Z 258.63,A -85,B 0,C 180,E1 -11132.609,E2 -11132.609} C_VEL
LIN {X 0,Y 397.124,Z 258.633,A -85,B 0,C 180,E1 -11135.981,E2 -11135.981} C_VEL
LIN {X 0,Y 397.134,Z 258.634,A -85,B 0,C 180,E1 -11139.704,E2 -11139.704} C_VEL
LIN {X 0,Y 397.177,Z 258.638,A -85,B 0,C 180,E1 -11142.844,E2 -11142.844} C_VEL
LIN {X 0,Y 397.221,Z 258.63,A -85,B 0,C 180,E1 -11146.678,E2 -11146.678} C_VEL
LIN {X 0,Y 397.212,Z 258.623,A -85,B 0,C 180,E1 -11149.808,E2 -11149.808} C_VEL
LIN {X 0,Y 397.347,Z 258.615,A -85,B 0,C 180,E1 -11152.888,E2 -11152.888} C_VEL
LIN {X 0,Y 397.249,Z 258.617,A -85,B 0,C 180,E1 -11154.925,E2 -11154.925} C_VEL
LIN {X 0,Y 397.445,Z 258.601,A -85,B 0,C 180,E1 -11157.973,E2 -11157.973} C_VEL
LIN {X 0,Y 397.574,Z 258.582,A -85,B 0,C 180,E1 -11160,E2 -11160} C_VEL
LIN {X 0,Y 397.375,Z 258.609,A -85,B 0,C 180,E1 -11163.041,E2 -11163.041} C_VEL
LIN {X 0,Y 397.357,Z 258.609,A -85,B 0,C 180,E1 -11167.112,E2 -11167.112} C_VEL
LIN {X 0,Y 397.211,Z 258.627,A -85,B 0,C 180,E1 -11170.191,E2 -11170.191} C_VEL
LIN {X 0,Y 397.22,Z 258.628,A -85,B 0,C 180,E1 -11173.321,E2 -11173.321} C_VEL
LIN {X 0,Y 397.175,Z 258.632,A -85,B 0,C 180,E1 -11177.155,E2 -11177.155} C_VEL
LIN {X 0,Y 397.096,Z 258.64,A -85,B 0,C 180,E1 -11180.73,E2 -11180.73} C_VEL
LIN {X 0,Y 397.126,Z 258.64,A -85,B 0,C 180,E1 -11184.018,E2 -11184.018} C_VEL
LIN {X 0,Y 397.189,Z 258.633,A -85,B 0,C 180,E1 -11187.39,E2 -11187.39} C_VEL
LIN {X 0,Y 397.078,Z 258.628,A -85,B 0,C 180,E1 -11190.882,E2 -11190.882} C_VEL
LIN {X 0,Y 397.12,Z 258.641,A -85,B 0,C 180,E1 -11194.494,E2 -11194.494} C_VEL
LIN {X 0,Y 397.102,Z 258.642,A -85,B 0,C 180,E1 -11198.275,E2 -11198.275} C_VEL
LIN {X 0,Y 397.084,Z 258.644,A -85,B 0,C 180,E1 -11200.909,E2 -11200.909} C_VEL
LIN {X 0,Y 397.097,Z 258.643,A -85,B 0,C 180,E1 -11203.649,E2 -11203.649} C_VEL
LIN {X 0,Y 397.098,Z 258.626,A -85,B 0,C 180,E1 -11206.521,E2 -11206.521} C_VEL
LIN {X 0,Y 397.111,Z 258.637,A -85,B 0,C 180,E1 -11210.423,E2 -11210.423} C_VEL
LIN {X 0,Y 397.105,Z 258.618,A -85,B 0,C 180,E1 -11214.266,E2 -11214.266} C_VEL
LIN {X 0,Y 397.112,Z 258.644,A -85,B 0,C 180,E1 -11216.728,E2 -11216.728} C_VEL
LIN {X 0,Y 397.138,Z 258.848,A -85,B 0,C 180,E1 -11219.049,E2 -11219.049} C_VEL
LIN {X 0,Y 400.399,Z 271.668,A -85,B 0,C 180,E1 -11221.712,E2 -11221.712} C_VEL
LIN {X 0,Y 403.188,Z 284.169,A -85,B 0,C 180,E1 -11224.166,E2 -11224.166} C_VEL
LIN {X 0,Y 402.586,Z 291.919,A -85,B 0,C 180,E1 -11225.506,E2 -11225.506} C_VEL
LIN {X 0,Y 402.004,Z 298.396,A -85,B 0,C 180,E1 -11226.554,E2 -11226.554} C_VEL
LIN {X 0,Y 405.572,Z 321.626,A -85,B 0,C 180,E1 -11227.218,E2 -11227.218} C_VEL
LIN {X 0,Y 403.687,Z 431.704,A -85,B 0,C 180,E1 -11229.291,E2 -11229.291} C_VEL
LIN {X 0,Y 403.053,Z 446.081,A -85,B 0,C 180,E1 -11229.757,E2 -11229.757} C_VEL
LIN {X 0,Y 402.339,Z 459.937,A -85,B 0,C 180,E1 -11230.418,E2 -11230.418} C_VEL
LIN {X 0,Y 401.522,Z 473.133,A -85,B 0,C 180,E1 -11231.26,E2 -11231.26} C_VEL
LIN {X 0,Y 400.55,Z 485.404,A -85,B 0,C 180,E1 -11232.251,E2 -11232.251} C_VEL
LIN {X 0,Y 399.542,Z 496.849,A -85,B 0,C 180,E1 -11233.391,E2 -11233.391} C_VEL
LIN {X 0,Y 398.587,Z 507.348,A -85,B 0,C 180,E1 -11234.664,E2 -11234.664} C_VEL
LIN {X 0,Y 397.794,Z 517.466,A -85,B 0,C 180,E1 -11236.155,E2 -11236.155} C_VEL
LIN {X 0,Y 397.127,Z 526.301,A -85,B 0,C 180,E1 -11237.739,E2 -11237.739} C_VEL
LIN {X 0,Y 396.476,Z 534.451,A -85,B 0,C 180,E1 -11239.532,E2 -11239.532} C_VEL
LIN {X 0,Y 396.119,Z 540.985,A -85,B 0,C 180,E1 -11241.326,E2 -11241.326} C_VEL
LIN {X 0,Y 395.923,Z 545.463,A -85,B 0,C 180,E1 -11242.862,E2 -11242.862} C_VEL
LIN {X 0,Y 395.78,Z 549.945,A -85,B 0,C 180,E1 -11244.906,E2 -11244.906} C_VEL
LIN {X 0,Y 395.723,Z 552.906,A -85,B 0,C 180,E1 -11246.946,E2 -11246.946} C_VEL
LIN {X 0,Y 395.789,Z 554.427,A -85,B 0,C 180,E1 -11248.983,E2 -11248.983} C_VEL
LIN {X 0,Y 395.789,Z 554.528,A -85,B 0,C 180,E1 -11251.017,E2 -11251.017} C_VEL
LIN {X 0,Y 395.721,Z 553.197,A -85,B 0,C 180,E1 -11253.054,E2 -11253.054} C_VEL
LIN {X 0,Y 395.794,Z 550.412,A -85,B 0,C 180,E1 -11255.094,E2 -11255.094} C_VEL
LIN {X 0,Y 395.924,Z 546.117,A -85,B 0,C 180,E1 -11257.138,E2 -11257.138} C_VEL
LIN {X 0,Y 396.261,Z 540.195,A -85,B 0,C 180,E1 -11259.185,E2 -11259.185} C_VEL
LIN {X 0,Y 396.693,Z 533.498,A -85,B 0,C 180,E1 -11260.979,E2 -11260.979} C_VEL
LIN {X 0,Y 397.382,Z 525.136,A -85,B 0,C 180,E1 -11262.772,E2 -11262.772} C_VEL
LIN {X 0,Y 398.167,Z 516.359,A -85,B 0,C 180,E1 -11264.306,E2 -11264.306} C_VEL
LIN {X 0,Y 399.098,Z 505.696,A -85,B 0,C 180,E1 -11265.84,E2 -11265.84} C_VEL
LIN {X 0,Y 400.236,Z 493.74,A -85,B 0,C 180,E1 -11267.236,E2 -11267.236} C_VEL
LIN {X 0,Y 401.371,Z 481.711,A -85,B 0,C 180,E1 -11268.371,E2 -11268.371} C_VEL
LIN {X 0,Y 402.401,Z 468.259,A -85,B 0,C 180,E1 -11269.38,E2 -11269.38} C_VEL
LIN {X 0,Y 403.302,Z 454.296,A -85,B 0,C 180,E1 -11270.177,E2 -11270.177} C_VEL
LIN {X 0,Y 404.078,Z 440.242,A -85,B 0,C 180,E1 -11270.755,E2 -11270.755} C_VEL
LIN {X 0,Y 404.589,Z 426.335,A -85,B 0,C 180,E1 -11271.127,E2 -11271.127} C_VEL
LIN {X 0,Y 406.361,Z 320.73,A -85,B 0,C 180,E1 -11273.112,E2 -11273.112} C_VEL
LIN {X 0,Y 402.557,Z 298.275,A -85,B 0,C 180,E1 -11273.811,E2 -11273.811} C_VEL
LIN {X 0,Y 403.724,Z 286.523,A -85,B 0,C 180,E1 -11275.797,E2 -11275.797} C_VEL
LIN {X 0,Y 402.362,Z 278.885,A -85,B 0,C 180,E1 -11277.29,E2 -11277.29} C_VEL
LIN {X 0,Y 398.548,Z 263.968,A -85,B 0,C 180,E1 -11280.392,E2 -11280.392} C_VEL
LIN {X 0,Y 397.115,Z 258.719,A -85,B 0,C 180,E1 -11281.584,E2 -11281.584} C_VEL
LIN {X 0,Y 397.123,Z 258.64,A -85,B 0,C 180,E1 -11284.493,E2 -11284.493} C_VEL
LIN {X 0,Y 397.099,Z 258.638,A -85,B 0,C 180,E1 -11288.275,E2 -11288.275} C_VEL
LIN {X 0,Y 397.151,Z 258.637,A -85,B 0,C 180,E1 -11291.993,E2 -11291.993} C_VEL
LIN {X 0,Y 397.109,Z 258.637,A -85,B 0,C 180,E1 -11295.065,E2 -11295.065} C_VEL
LIN {X 0,Y 397.063,Z 258.641,A -85,B 0,C 180,E1 -11298.021,E2 -11298.021} C_VEL
LIN {X 0,Y 397.129,Z 258.641,A -85,B 0,C 180,E1 -11301.138,E2 -11301.138} C_VEL
LIN {X 0,Y 397.115,Z 258.629,A -85,B 0,C 180,E1 -11304.496,E2 -11304.496} C_VEL
LIN {X 0,Y 397.076,Z 258.646,A -85,B 0,C 180,E1 -11307.928,E2 -11307.928} C_VEL
LIN {X 0,Y 397.121,Z 258.628,A -85,B 0,C 180,E1 -11311.457,E2 -11311.457} C_VEL
LIN {X 0,Y 397.147,Z 258.636,A -85,B 0,C 180,E1 -11314.487,E2 -11314.487} C_VEL
LIN {X 0,Y 397.103,Z 258.643,A -85,B 0,C 180,E1 -11317.086,E2 -11317.086} C_VEL
LIN {X 0,Y 397.142,Z 258.639,A -85,B 0,C 180,E1 -11320.353,E2 -11320.353} C_VEL
LIN {X 0,Y 397.16,Z 258.633,A -85,B 0,C 180,E1 -11323.553,E2 -11323.553} C_VEL
LIN {X 0,Y 397.223,Z 258.626,A -85,B 0,C 180,E1 -11326.703,E2 -11326.703} C_VEL
LIN {X 0,Y 397.212,Z 258.632,A -85,B 0,C 180,E1 -11329.809,E2 -11329.809} C_VEL
LIN {X 0,Y 397.346,Z 258.604,A -85,B 0,C 180,E1 -11332.888,E2 -11332.888} C_VEL
LIN {X 0,Y 397.25,Z 258.625,A -85,B 0,C 180,E1 -11334.925,E2 -11334.925} C_VEL
LIN {X 0,Y 397.446,Z 258.598,A -85,B 0,C 180,E1 -11337.974,E2 -11337.974} C_VEL
LIN {X 0,Y 397.574,Z 258.585,A -85,B 0,C 180,E1 -11340,E2 -11340} C_VEL
LIN {X 0,Y 397.376,Z 258.603,A -85,B 0,C 180,E1 -11343.042,E2 -11343.042} C_VEL
LIN {X 0,Y 397.358,Z 258.606,A -85,B 0,C 180,E1 -11347.112,E2 -11347.112} C_VEL
LIN {X 0,Y 397.212,Z 258.627,A -85,B 0,C 180,E1 -11350.192,E2 -11350.192} C_VEL
LIN {X 0,Y 397.222,Z 258.631,A -85,B 0,C 180,E1 -11353.322,E2 -11353.322} C_VEL
LIN {X 0,Y 397.177,Z 258.634,A -85,B 0,C 180,E1 -11357.156,E2 -11357.156} C_VEL
LIN {X 0,Y 397.104,Z 258.639,A -85,B 0,C 180,E1 -11360.73,E2 -11360.73} C_VEL
LIN {X 0,Y 397.129,Z 258.636,A -85,B 0,C 180,E1 -11364.019,E2 -11364.019} C_VEL
LIN {X 0,Y 397.191,Z 258.624,A -85,B 0,C 180,E1 -11367.391,E2 -11367.391} C_VEL
LIN {X 0,Y 397.076,Z 258.642,A -85,B 0,C 180,E1 -11370.883,E2 -11370.883} C_VEL
LIN {X 0,Y 397.124,Z 258.63,A -85,B 0,C 180,E1 -11374.494,E2 -11374.494} C_VEL
LIN {X 0,Y 397.102,Z 258.645,A -85,B 0,C 180,E1 -11378.276,E2 -11378.276} C_VEL
LIN {X 0,Y 397.087,Z 258.638,A -85,B 0,C 180,E1 -11380.91,E2 -11380.91} C_VEL
LIN {X 0,Y 397.1,Z 258.637,A -85,B 0,C 180,E1 -11383.649,E2 -11383.649} C_VEL
LIN {X 0,Y 397.105,Z 258.646,A -85,B 0,C 180,E1 -11386.521,E2 -11386.521} C_VEL
LIN {X 0,Y 397.115,Z 258.627,A -85,B 0,C 180,E1 -11390.424,E2 -11390.424} C_VEL
LIN {X 0,Y 397.109,Z 258.645,A -85,B 0,C 180,E1 -11394.266,E2 -11394.266} C_VEL
LIN {X 0,Y 397.121,Z 258.79,A -85,B 0,C 180,E1 -11395.994,E2 -11395.994} C_VEL
LIN {X 0,Y 400.1,Z 270.723,A -85,B 0,C 180,E1 -11398.791,E2 -11398.791} C_VEL
LIN {X 0,Y 402.706,Z 282.365,A -85,B 0,C 180,E1 -11401.369,E2 -11401.369} C_VEL
LIN {X 0,Y 402.796,Z 286.37,A -85,B 0,C 180,E1 -11402.178,E2 -11402.178} C_VEL
LIN {X 0,Y 401.009,Z 305.528,A -85,B 0,C 180,E1 -11405.828,E2 -11405.828} C_VEL
LIN {X 0,Y 400.49,Z 312.77,A -85,B 0,C 180,E1 -11407.137,E2 -11407.137} C_VEL
LIN {X 0,Y 405.547,Z 340.167,A -85,B 0,C 180,E1 -11407.942,E2 -11407.942} C_VEL
LIN {X 0,Y 404.492,Z 425.813,A -85,B 0,C 180,E1 -11409.4,E2 -11409.4} C_VEL
LIN {X 0,Y 403.958,Z 439.102,A -85,B 0,C 180,E1 -11409.817,E2 -11409.817} C_VEL
LIN {X 0,Y 403.35,Z 452.503,A -85,B 0,C 180,E1 -11410.467,E2 -11410.467} C_VEL
LIN {X 0,Y 402.433,Z 464.825,A -85,B 0,C 180,E1 -11411.283,E2 -11411.283} C_VEL
LIN {X 0,Y 401.329,Z 476.416,A -85,B 0,C 180,E1 -11412.286,E2 -11412.286} C_VEL
LIN {X 0,Y 400.227,Z 486.84,A -85,B 0,C 180,E1 -11413.42,E2 -11413.42} C_VEL
LIN {X 0,Y 399.238,Z 496.254,A -85,B 0,C 180,E1 -11414.69,E2 -11414.69} C_VEL
LIN {X 0,Y 398.337,Z 504.336,A -85,B 0,C 180,E1 -11416.024,E2 -11416.024} C_VEL
LIN {X 0,Y 397.667,Z 511.586,A -85,B 0,C 180,E1 -11417.497,E2 -11417.497} C_VEL
LIN {X 0,Y 396.857,Z 518.583,A -85,B 0,C 180,E1 -11419.284,E2 -11419.284} C_VEL
LIN {X 0,Y 396.442,Z 523.281,A -85,B 0,C 180,E1 -11420.819,E2 -11420.819} C_VEL
LIN {X 0,Y 396.157,Z 526.92,A -85,B 0,C 180,E1 -11422.354,E2 -11422.354} C_VEL
LIN {X 0,Y 395.913,Z 529.601,A -85,B 0,C 180,E1 -11423.886,E2 -11423.886} C_VEL
LIN {X 0,Y 395.792,Z 531.778,A -85,B 0,C 180,E1 -11425.927,E2 -11425.927} C_VEL
LIN {X 0,Y 395.814,Z 532.482,A -85,B 0,C 180,E1 -11427.965,E2 -11427.965} C_VEL
LIN {X 0,Y 395.783,Z 531.681,A -85,B 0,C 180,E1 -11430,E2 -11430} C_VEL
LIN {X 0,Y 395.857,Z 530.225,A -85,B 0,C 180,E1 -11431.416,E2 -11431.416} C_VEL
LIN {X 0,Y 395.275,Z 529.121,A -85,B 0,C 180,E1 -11432.252,E2 -11432.252} C_VEL
LIN {X 0,Y 392.56,Z 526.817,A -85,B 0,C 180,E1 -11433.602,E2 -11433.602} C_VEL
LIN {X 0,Y 390.315,Z 524.534,A -85,B 0,C 180,E1 -11434.672,E2 -11434.672} C_VEL
LIN {X 0,Y 389.462,Z 522.44,A -85,B 0,C 180,E1 -11435.478,E2 -11435.478} C_VEL
LIN {X 0,Y 389.454,Z 521.651,A -85,B 0,C 180,E1 -11435.746,E2 -11435.746} C_VEL
LIN {X 0,Y 389.897,Z 516.685,A -85,B 0,C 180,E1 -11437.249,E2 -11437.249} C_VEL
LIN {X 0,Y 390.627,Z 509.1,A -85,B 0,C 180,E1 -11439.057,E2 -11439.057} C_VEL
LIN {X 0,Y 391.541,Z 500.938,A -85,B 0,C 180,E1 -11440.602,E2 -11440.602} C_VEL
LIN {X 0,Y 392.431,Z 492.591,A -85,B 0,C 180,E1 -11441.885,E2 -11441.885} C_VEL
LIN {X 0,Y 393.329,Z 482.346,A -85,B 0,C 180,E1 -11443.168,E2 -11443.168} C_VEL
LIN {X 0,Y 394.295,Z 472.242,A -85,B 0,C 180,E1 -11444.186,E2 -11444.186} C_VEL
LIN {X 0,Y 395.118,Z 462.985,A -85,B 0,C 180,E1 -11444.946,E2 -11444.946} C_VEL
LIN {X 0,Y 395.89,Z 451.29,A -85,B 0,C 180,E1 -11445.707,E2 -11445.707} C_VEL
LIN {X 0,Y 396.634,Z 437.948,A -85,B 0,C 180,E1 -11446.337,E2 -11446.337} C_VEL
LIN {X 0,Y 397.037,Z 425.903,A -85,B 0,C 180,E1 -11446.712,E2 -11446.712} C_VEL
LIN {X 0,Y 398.073,Z 340.834,A -85,B 0,C 180,E1 -11448.179,E2 -11448.179} C_VEL
LIN {X 0,Y 393.224,Z 312.833,A -85,B 0,C 180,E1 -11448.968,E2 -11448.968} C_VEL
LIN {X 0,Y 393.206,Z 311.949,A -85,B 0,C 180,E1 -11449.065,E2 -11449.065} C_VEL
LIN {X 0,Y 394.713,Z 293.886,A -85,B 0,C 180,E1 -11452.507,E2 -11452.507} C_VEL
LIN {X 0,Y 395.57,Z 284.157,A -85,B 0,C 180,E1 -11454.396,E2 -11454.396} C_VEL
LIN {X 0,Y 392.722,Z 270.296,A -85,B 0,C 180,E1 -11457.439,E2 -11457.439} C_VEL
LIN {X 0,Y 390.079,Z 259.62,A -85,B 0,C 180,E1 -11459.943,E2 -11459.943} C_VEL
LIN {X 0,Y 390.069,Z 259.497,A -85,B 0,C 180,E1 -11463.954,E2 -11463.954} C_VEL
LIN {X 0,Y 390.044,Z 259.519,A -85,B 0,C 180,E1 -11467.55,E2 -11467.55} C_VEL
LIN {X 0,Y 390.057,Z 259.515,A -85,B 0,C 180,E1 -11470.82,E2 -11470.82} C_VEL
LIN {X 0,Y 390.056,Z 259.518,A -85,B 0,C 180,E1 -11473.886,E2 -11473.886} C_VEL
LIN {X 0,Y 390.056,Z 259.52,A -85,B 0,C 180,E1 -11476.789,E2 -11476.789} C_VEL
LIN {X 0,Y 390.054,Z 259.506,A -85,B 0,C 180,E1 -11479.56,E2 -11479.56} C_VEL
LIN {X 0,Y 390.042,Z 259.522,A -85,B 0,C 180,E1 -11482.448,E2 -11482.448} C_VEL
LIN {X 0,Y 390.065,Z 259.5,A -85,B 0,C 180,E1 -11485.975,E2 -11485.975} C_VEL
LIN {X 0,Y 390.049,Z 259.522,A -85,B 0,C 180,E1 -11489.867,E2 -11489.867} C_VEL
LIN {X 0,Y 390.11,Z 259.517,A -85,B 0,C 180,E1 -11493.231,E2 -11493.231} C_VEL
LIN {X 0,Y 390.072,Z 259.517,A -85,B 0,C 180,E1 -11496.76,E2 -11496.76} C_VEL
LIN {X 0,Y 390.099,Z 259.51,A -85,B 0,C 180,E1 -11499.982,E2 -11499.982} C_VEL
LIN {X 0,Y 390.133,Z 259.511,A -85,B 0,C 180,E1 -11503.248,E2 -11503.248} C_VEL
LIN {X 0,Y 390.189,Z 259.504,A -85,B 0,C 180,E1 -11506.561,E2 -11506.561} C_VEL
LIN {X 0,Y 390.199,Z 259.499,A -85,B 0,C 180,E1 -11510.671,E2 -11510.671} C_VEL
LIN {X 0,Y 390.321,Z 259.487,A -85,B 0,C 180,E1 -11513.798,E2 -11513.798} C_VEL
LIN {X 0,Y 390.414,Z 259.477,A -85,B 0,C 180,E1 -11517.936,E2 -11517.936} C_VEL
LIN {X 0,Y 390.543,Z 259.458,A -85,B 0,C 180,E1 -11520,E2 -11520} C_VEL
LIN {X 0,Y 390.309,Z 259.489,A -85,B 0,C 180,E1 -11523.096,E2 -11523.096} C_VEL
LIN {X 0,Y 390.323,Z 259.481,A -85,B 0,C 180,E1 -11526.202,E2 -11526.202} C_VEL
LIN {X 0,Y 390.308,Z 259.493,A -85,B 0,C 180,E1 -11528.282,E2 -11528.282} C_VEL
LIN {X 0,Y 390.164,Z 259.509,A -85,B 0,C 180,E1 -11532.483,E2 -11532.483} C_VEL
LIN {X 0,Y 390.132,Z 259.508,A -85,B 0,C 180,E1 -11535.677,E2 -11535.677} C_VEL
LIN {X 0,Y 390.099,Z 259.515,A -85,B 0,C 180,E1 -11538.922,E2 -11538.922} C_VEL
LIN {X 0,Y 390.034,Z 259.528,A -85,B 0,C 180,E1 -11542.234,E2 -11542.234} C_VEL
LIN {X 0,Y 390.113,Z 259.512,A -85,B 0,C 180,E1 -11545.744,E2 -11545.744} C_VEL
LIN {X 0,Y 390.06,Z 259.511,A -85,B 0,C 180,E1 -11549.109,E2 -11549.109} C_VEL
LIN {X 0,Y 390.038,Z 259.523,A -85,B 0,C 180,E1 -11552.722,E2 -11552.722} C_VEL
LIN {X 0,Y 390.052,Z 259.511,A -85,B 0,C 180,E1 -11555.826,E2 -11555.826} C_VEL
LIN {X 0,Y 390.067,Z 259.521,A -85,B 0,C 180,E1 -11559.219,E2 -11559.219} C_VEL
LIN {X 0,Y 390.038,Z 259.514,A -85,B 0,C 180,E1 -11562.375,E2 -11562.375} C_VEL
LIN {X 0,Y 390.041,Z 259.521,A -85,B 0,C 180,E1 -11565.355,E2 -11565.355} C_VEL
LIN {X 0,Y 390.026,Z 259.485,A -85,B 0,C 180,E1 -11568.187,E2 -11568.187} C_VEL
LIN {X 0,Y 390.088,Z 259.518,A -85,B 0,C 180,E1 -11570.908,E2 -11570.908} C_VEL
LIN {X 0,Y 390.082,Z 259.495,A -85,B 0,C 180,E1 -11574.794,E2 -11574.794} C_VEL
LIN {X 0,Y 390.09,Z 259.71,A -85,B 0,C 180,E1 -11578.606,E2 -11578.606} C_VEL
LIN {X 0,Y 393.428,Z 272.779,A -85,B 0,C 180,E1 -11581.39,E2 -11581.39} C_VEL
LIN {X 0,Y 396.334,Z 285.62,A -85,B 0,C 180,E1 -11583.968,E2 -11583.968} C_VEL
LIN {X 0,Y 396.025,Z 290.49,A -85,B 0,C 180,E1 -11584.832,E2 -11584.832} C_VEL
LIN {X 0,Y 395.273,Z 298.571,A -85,B 0,C 180,E1 -11586.178,E2 -11586.178} C_VEL
LIN {X 0,Y 398.934,Z 322.429,A -85,B 0,C 180,E1 -11586.874,E2 -11586.874} C_VEL
LIN {X 0,Y 396.99,Z 431.453,A -85,B 0,C 180,E1 -11588.959,E2 -11588.959} C_VEL
LIN {X 0,Y 396.334,Z 445.896,A -85,B 0,C 180,E1 -11589.432,E2 -11589.432} C_VEL
LIN {X 0,Y 395.537,Z 460.341,A -85,B 0,C 180,E1 -11590.135,E2 -11590.135} C_VEL
LIN {X 0,Y 394.718,Z 473.162,A -85,B 0,C 180,E1 -11590.971,E2 -11590.971} C_VEL
LIN {X 0,Y 393.743,Z 484.901,A -85,B 0,C 180,E1 -11591.933,E2 -11591.933} C_VEL
LIN {X 0,Y 392.662,Z 496.409,A -85,B 0,C 180,E1 -11593.092,E2 -11593.092} C_VEL
LIN {X 0,Y 391.667,Z 506.959,A -85,B 0,C 180,E1 -11594.386,E2 -11594.386} C_VEL
LIN {X 0,Y 390.815,Z 517.405,A -85,B 0,C 180,E1 -11595.951,E2 -11595.951} C_VEL
LIN {X 0,Y 390.114,Z 525.995,A -85,B 0,C 180,E1 -11597.515,E2 -11597.515} C_VEL
LIN {X 0,Y 389.459,Z 534.171,A -85,B 0,C 180,E1 -11599.341,E2 -11599.341} C_VEL
LIN {X 0,Y 389.059,Z 540.724,A -85,B 0,C 180,E1 -11601.168,E2 -11601.168} C_VEL
LIN {X 0,Y 388.817,Z 546.499,A -85,B 0,C 180,E1 -11603.253,E2 -11603.253} C_VEL
LIN {X 0,Y 388.681,Z 549.715,A -85,B 0,C 180,E1 -11604.813,E2 -11604.813} C_VEL
LIN {X 0,Y 388.68,Z 551.388,A -85,B 0,C 180,E1 -11605.852,E2 -11605.852} C_VEL
LIN {X 0,Y 388.659,Z 553.633,A -85,B 0,C 180,E1 -11607.928,E2 -11607.928} C_VEL
LIN {X 0,Y 388.706,Z 554.453,A -85,B 0,C 180,E1 -11610,E2 -11610} C_VEL
LIN {X 0,Y 388.658,Z 553.852,A -85,B 0,C 180,E1 -11612.073,E2 -11612.073} C_VEL
LIN {X 0,Y 388.682,Z 551.805,A -85,B 0,C 180,E1 -11614.148,E2 -11614.148} C_VEL
LIN {X 0,Y 388.775,Z 548.283,A -85,B 0,C 180,E1 -11616.227,E2 -11616.227} C_VEL
LIN {X 0,Y 388.992,Z 543.195,A -85,B 0,C 180,E1 -11618.31,E2 -11618.31} C_VEL
LIN {X 0,Y 389.317,Z 538.255,A -85,B 0,C 180,E1 -11619.875,E2 -11619.875} C_VEL
LIN {X 0,Y 389.93,Z 531.101,A -85,B 0,C 180,E1 -11621.699,E2 -11621.699} C_VEL
LIN {X 0,Y 390.582,Z 523.592,A -85,B 0,C 180,E1 -11623.263,E2 -11623.263} C_VEL
LIN {X 0,Y 391.371,Z 514.54,A -85,B 0,C 180,E1 -11624.826,E2 -11624.826} C_VEL
LIN {X 0,Y 392.231,Z 505.528,A -85,B 0,C 180,E1 -11626.124,E2 -11626.124} C_VEL
LIN {X 0,Y 393.431,Z 493.568,A -85,B 0,C 180,E1 -11627.544,E2 -11627.544} C_VEL
LIN {X 0,Y 394.629,Z 481.53,A -85,B 0,C 180,E1 -11628.697,E2 -11628.697} C_VEL
LIN {X 0,Y 395.565,Z 469.501,A -85,B 0,C 180,E1 -11629.627,E2 -11629.627} C_VEL
LIN {X 0,Y 396.492,Z 456.251,A -85,B 0,C 180,E1 -11630.424,E2 -11630.424} C_VEL
LIN {X 0,Y 397.326,Z 442.636,A -85,B 0,C 180,E1 -11631.022,E2 -11631.022} C_VEL
LIN {X 0,Y 397.9,Z 428.78,A -85,B 0,C 180,E1 -11631.432,E2 -11631.432} C_VEL
LIN {X 0,Y 399.828,Z 322.172,A -85,B 0,C 180,E1 -11633.472,E2 -11633.472} C_VEL
LIN {X 0,Y 395.86,Z 298.457,A -85,B 0,C 180,E1 -11634.222,E2 -11634.222} C_VEL
LIN {X 0,Y 396.959,Z 288.145,A -85,B 0,C 180,E1 -11635.988,E2 -11635.988} C_VEL
LIN {X 0,Y 395.125,Z 278.981,A -85,B 0,C 180,E1 -11637.833,E2 -11637.833} C_VEL
LIN {X 0,Y 391.837,Z 266.072,A -85,B 0,C 180,E1 -11640.579,E2 -11640.579} C_VEL
LIN {X 0,Y 390.062,Z 259.592,A -85,B 0,C 180,E1 -11642.077,E2 -11642.077} C_VEL
LIN {X 0,Y 390.082,Z 259.499,A -85,B 0,C 180,E1 -11645.206,E2 -11645.206} C_VEL
LIN {X 0,Y 390.066,Z 259.523,A -85,B 0,C 180,E1 -11649.218,E2 -11649.218} C_VEL
LIN {X 0,Y 390.118,Z 259.518,A -85,B 0,C 180,E1 -11652.386,E2 -11652.386} C_VEL
LIN {X 0,Y 390.059,Z 259.517,A -85,B 0,C 180,E1 -11655.357,E2 -11655.357} C_VEL
LIN {X 0,Y 390.027,Z 259.515,A -85,B 0,C 180,E1 -11658.186,E2 -11658.186} C_VEL
LIN {X 0,Y 390.088,Z 259.519,A -85,B 0,C 180,E1 -11660.908,E2 -11660.908} C_VEL
LIN {X 0,Y 390.081,Z 259.507,A -85,B 0,C 180,E1 -11664.793,E2 -11664.793} C_VEL
LIN {X 0,Y 390.022,Z 259.517,A -85,B 0,C 180,E1 -11668.496,E2 -11668.496} C_VEL
LIN {X 0,Y 390.112,Z 259.507,A -85,B 0,C 180,E1 -11672.07,E2 -11672.07} C_VEL
LIN {X 0,Y 390.074,Z 259.516,A -85,B 0,C 180,E1 -11675.519,E2 -11675.519} C_VEL
LIN {X 0,Y 390.05,Z 259.518,A -85,B 0,C 180,E1 -11678.878,E2 -11678.878} C_VEL
LIN {X 0,Y 390.122,Z 259.513,A -85,B 0,C 180,E1 -11682.167,E2 -11682.167} C_VEL
LIN {X 0,Y 390.138,Z 259.51,A -85,B 0,C 180,E1 -11685.393,E2 -11685.393} C_VEL
LIN {X 0,Y 390.142,Z 259.504,A -85,B 0,C 180,E1 -11688.571,E2 -11688.571} C_VEL
LIN {X 0,Y 390.302,Z 259.484,A -85,B 0,C 180,E1 -11692.032,E2 -11692.032} C_VEL
LIN {X 0,Y 390.221,Z 259.5,A -85,B 0,C 180,E1 -11694.834,E2 -11694.834} C_VEL
LIN {X 0,Y 390.414,Z 259.473,A -85,B 0,C 180,E1 -11697.937,E2 -11697.937} C_VEL
LIN {X 0,Y 390.544,Z 259.461,A -85,B 0,C 180,E1 -11700,E2 -11700} C_VEL
LIN {X 0,Y 390.31,Z 259.484,A -85,B 0,C 180,E1 -11703.097,E2 -11703.097} C_VEL
LIN {X 0,Y 390.304,Z 259.483,A -85,B 0,C 180,E1 -11706.648,E2 -11706.648} C_VEL
LIN {X 0,Y 390.2,Z 259.507,A -85,B 0,C 180,E1 -11709.329,E2 -11709.329} C_VEL
LIN {X 0,Y 390.19,Z 259.509,A -85,B 0,C 180,E1 -11713.439,E2 -11713.439} C_VEL
LIN {X 0,Y 390.144,Z 259.512,A -85,B 0,C 180,E1 -11717.308,E2 -11717.308} C_VEL
LIN {X 0,Y 390.084,Z 259.512,A -85,B 0,C 180,E1 -11720.471,E2 -11720.471} C_VEL
LIN {X 0,Y 390.086,Z 259.515,A -85,B 0,C 180,E1 -11723.352,E2 -11723.352} C_VEL
LIN {X 0,Y 390.11,Z 259.515,A -85,B 0,C 180,E1 -11726.769,E2 -11726.769} C_VEL
LIN {X 0,Y 390.036,Z 259.514,A -85,B 0,C 180,E1 -11730.301,E2 -11730.301} C_VEL
LIN {X 0,Y 390.066,Z 259.513,A -85,B 0,C 180,E1 -11734.025,E2 -11734.025} C_VEL
LIN {X 0,Y 390.043,Z 259.524,A -85,B 0,C 180,E1 -11737.552,E2 -11737.552} C_VEL
LIN {X 0,Y 390.055,Z 259.512,A -85,B 0,C 180,E1 -11740.822,E2 -11740.822} C_VEL
LIN {X 0,Y 390.054,Z 259.513,A -85,B 0,C 180,E1 -11743.887,E2 -11743.887} C_VEL
LIN {X 0,Y 390.059,Z 259.519,A -85,B 0,C 180,E1 -11746.791,E2 -11746.791} C_VEL
LIN {X 0,Y 390.058,Z 259.522,A -85,B 0,C 180,E1 -11749.562,E2 -11749.562} C_VEL
LIN {X 0,Y 390.044,Z 259.497,A -85,B 0,C 180,E1 -11752.45,E2 -11752.45} C_VEL
LIN {X 0,Y 390.109,Z 259.712,A -85,B 0,C 180,E1 -11755.544,E2 -11755.544} C_VEL
LIN {X 0,Y 393.187,Z 271.992,A -85,B 0,C 180,E1 -11758.478,E2 -11758.478} C_VEL
LIN {X 0,Y 395.757,Z 283.571,A -85,B 0,C 180,E1 -11761.094,E2 -11761.094} C_VEL
LIN {X 0,Y 396.128,Z 286.243,A -85,B 0,C 180,E1 -11761.668,E2 -11761.668} C_VEL
LIN {X 0,Y 394.414,Z 304.017,A -85,B 0,C 180,E1 -11765.122,E2 -11765.122} C_VEL
LIN {X 0,Y 393.678,Z 312.49,A -85,B 0,C 180,E1 -11766.701,E2 -11766.701} C_VEL
LIN {X 0,Y 398.907,Z 340.618,A -85,B 0,C 180,E1 -11767.56,E2 -11767.56} C_VEL
LIN {X 0,Y 398.868,Z 357.534,A -85,B 0,C 180,E1 -11767.861,E2 -11767.861} C_VEL
LIN {X 0,Y 397.876,Z 425.953,A -85,B 0,C 180,E1 -11769.042,E2 -11769.042} C_VEL
LIN {X 0,Y 397.295,Z 439.488,A -85,B 0,C 180,E1 -11769.475,E2 -11769.475} C_VEL
LIN {X 0,Y 396.702,Z 452.187,A -85,B 0,C 180,E1 -11770.101,E2 -11770.101} C_VEL
LIN {X 0,Y 395.826,Z 463.225,A -85,B 0,C 180,E1 -11770.824,E2 -11770.824} C_VEL
LIN {X 0,Y 394.88,Z 473.902,A -85,B 0,C 180,E1 -11771.719,E2 -11771.719} C_VEL
LIN {X 0,Y 393.686,Z 484.835,A -85,B 0,C 180,E1 -11772.869,E2 -11772.869} C_VEL
LIN {X 0,Y 392.586,Z 494.615,A -85,B 0,C 180,E1 -11774.157,E2 -11774.157} C_VEL
LIN {X 0,Y 391.507,Z 503.805,A -85,B 0,C 180,E1 -11775.655,E2 -11775.655} C_VEL
LIN {X 0,Y 390.716,Z 511.721,A -85,B 0,C 180,E1 -11777.271,E2 -11777.271} C_VEL
LIN {X 0,Y 389.854,Z 518.727,A -85,B 0,C 180,E1 -11779.089,E2 -11779.089} C_VEL
LIN {X 0,Y 389.393,Z 523.434,A -85,B 0,C 180,E1 -11780.652,E2 -11780.652} C_VEL
LIN {X 0,Y 389.087,Z 527.083,A -85,B 0,C 180,E1 -11782.214,E2 -11782.214} C_VEL
LIN {X 0,Y 388.837,Z 529.774,A -85,B 0,C 180,E1 -11783.774,E2 -11783.774} C_VEL
LIN {X 0,Y 388.716,Z 531.961,A -85,B 0,C 180,E1 -11785.853,E2 -11785.853} C_VEL
LIN {X 0,Y 388.713,Z 532.683,A -85,B 0,C 180,E1 -11787.928,E2 -11787.928} C_VEL
LIN {X 0,Y 388.712,Z 531.896,A -85,B 0,C 180,E1 -11790,E2 -11790} C_VEL
LIN {X 0,Y 388.879,Z 529.657,A -85,B 0,C 180,E1 -11792.071,E2 -11792.071} C_VEL
LIN {X 0,Y 389.143,Z 526.925,A -85,B 0,C 180,E1 -11793.624,E2 -11793.624} C_VEL
LIN {X 0,Y 389.276,Z 523.249,A -85,B 0,C 180,E1 -11795.179,E2 -11795.179} C_VEL
LIN {X 0,Y 389.454,Z 521.651,A -85,B 0,C 180,E1 -11795.746,E2 -11795.746} C_VEL
LIN {X 0,Y 389.023,Z 519.243,A -85,B 0,C 180,E1 -11796.536,E2 -11796.536} C_VEL
LIN {X 0,Y 386.574,Z 514.968,A -85,B 0,C 180,E1 -11797.812,E2 -11797.812} C_VEL
LIN {X 0,Y 384.215,Z 510.129,A -85,B 0,C 180,E1 -11799.053,E2 -11799.053} C_VEL
LIN {X 0,Y 383.925,Z 506.76,A -85,B 0,C 180,E1 -11799.777,E2 -11799.777} C_VEL
LIN {X 0,Y 384.924,Z 498.147,A -85,B 0,C 180,E1 -11801.319,E2 -11801.319} C_VEL
LIN {X 0,Y 385.994,Z 488.2,A -85,B 0,C 180,E1 -11802.754,E2 -11802.754} C_VEL
LIN {X 0,Y 386.937,Z 478.08,A -85,B 0,C 180,E1 -11803.925,E2 -11803.925} C_VEL
LIN {X 0,Y 387.936,Z 466.893,A -85,B 0,C 180,E1 -11804.96,E2 -11804.96} C_VEL
LIN {X 0,Y 388.791,Z 456.311,A -85,B 0,C 180,E1 -11805.732,E2 -11805.732} C_VEL
LIN {X 0,Y 389.642,Z 443.558,A -85,B 0,C 180,E1 -11806.436,E2 -11806.436} C_VEL
LIN {X 0,Y 390.178,Z 431.068,A -85,B 0,C 180,E1 -11806.915,E2 -11806.915} C_VEL
LIN {X 0,Y 390.517,Z 415.387,A -85,B 0,C 180,E1 -11807.257,E2 -11807.257} C_VEL
LIN {X 0,Y 391.448,Z 341.784,A -85,B 0,C 180,E1 -11808.529,E2 -11808.529} C_VEL
LIN {X 0,Y 386.409,Z 312.563,A -85,B 0,C 180,E1 -11809.376,E2 -11809.376} C_VEL
LIN {X 0,Y 386.578,Z 309.343,A -85,B 0,C 180,E1 -11809.93,E2 -11809.93} C_VEL
LIN {X 0,Y 388.218,Z 291.21,A -85,B 0,C 180,E1 -11813.47,E2 -11813.47} C_VEL
LIN {X 0,Y 388.73,Z 285.647,A -85,B 0,C 180,E1 -11814.571,E2 -11814.571} C_VEL
LIN {X 0,Y 385.837,Z 271.784,A -85,B 0,C 180,E1 -11817.676,E2 -11817.676} C_VEL
LIN {X 0,Y 383.018,Z 260.527,A -85,B 0,C 180,E1 -11820.369,E2 -11820.369} C_VEL
LIN {X 0,Y 383.005,Z 260.377,A -85,B 0,C 180,E1 -11823.4,E2 -11823.4} C_VEL
LIN {X 0,Y 383.033,Z 260.4,A -85,B 0,C 180,E1 -11826.164,E2 -11826.164} C_VEL
LIN {X 0,Y 383.009,Z 260.398,A -85,B 0,C 180,E1 -11829.957,E2 -11829.957} C_VEL
LIN {X 0,Y 383.005,Z 260.401,A -85,B 0,C 180,E1 -11832.778,E2 -11832.778} C_VEL
LIN {X 0,Y 382.997,Z 260.393,A -85,B 0,C 180,E1 -11835.788,E2 -11835.788} C_VEL
LIN {X 0,Y 382.986,Z 260.397,A -85,B 0,C 180,E1 -11838.795,E2 -11838.795} C_VEL
LIN {X 0,Y 382.998,Z 260.399,A -85,B 0,C 180,E1 -11842.095,E2 -11842.095} C_VEL
LIN {X 0,Y 383.015,Z 260.381,A -85,B 0,C 180,E1 -11845.331,E2 -11845.331} C_VEL
LIN {X 0,Y 382.983,Z 260.404,A -85,B 0,C 180,E1 -11849.081,E2 -11849.081} C_VEL
LIN {X 0,Y 383.053,Z 260.391,A -85,B 0,C 180,E1 -11852.697,E2 -11852.697} C_VEL
LIN {X 0,Y 383.046,Z 260.391,A -85,B 0,C 180,E1 -11855.039,E2 -11855.039} C_VEL
LIN {X 0,Y 382.993,Z 260.403,A -85,B 0,C 180,E1 -11858.469,E2 -11858.469} C_VEL
LIN {X 0,Y 383.058,Z 260.391,A -85,B 0,C 180,E1 -11861.826,E2 -11861.826} C_VEL
LIN {X 0,Y 383.107,Z 260.381,A -85,B 0,C 180,E1 -11865.118,E2 -11865.118} C_VEL
LIN {X 0,Y 383.092,Z 260.392,A -85,B 0,C 180,E1 -11868.357,E2 -11868.357} C_VEL
LIN {X 0,Y 383.258,Z 260.366,A -85,B 0,C 180,E1 -11871.975,E2 -11871.975} C_VEL
LIN {X 0,Y 383.193,Z 260.369,A -85,B 0,C 180,E1 -11874.738,E2 -11874.738} C_VEL
LIN {X 0,Y 383.381,Z 260.353,A -85,B 0,C 180,E1 -11877.899,E2 -11877.899} C_VEL
LIN {X 0,Y 383.513,Z 260.333,A -85,B 0,C 180,E1 -11880,E2 -11880} C_VEL
LIN {X 0,Y 383.245,Z 260.369,A -85,B 0,C 180,E1 -11883.153,E2 -11883.153} C_VEL
LIN {X 0,Y 383.28,Z 260.359,A -85,B 0,C 180,E1 -11886.316,E2 -11886.316} C_VEL
LIN {X 0,Y 383.253,Z 260.372,A -85,B 0,C 180,E1 -11888.436,E2 -11888.436} C_VEL
LIN {X 0,Y 383.09,Z 260.381,A -85,B 0,C 180,E1 -11891.642,E2 -11891.642} C_VEL
LIN {X 0,Y 383.103,Z 260.383,A -85,B 0,C 180,E1 -11894.882,E2 -11894.882} C_VEL
LIN {X 0,Y 383.083,Z 260.394,A -85,B 0,C 180,E1 -11898.172,E2 -11898.172} C_VEL
LIN {X 0,Y 382.987,Z 260.398,A -85,B 0,C 180,E1 -11901.531,E2 -11901.531} C_VEL
LIN {X 0,Y 383.046,Z 260.389,A -85,B 0,C 180,E1 -11904.96,E2 -11904.96} C_VEL
LIN {X 0,Y 383.044,Z 260.387,A -85,B 0,C 180,E1 -11908.492,E2 -11908.492} C_VEL
LIN {X 0,Y 383.005,Z 260.392,A -85,B 0,C 180,E1 -11912.15,E2 -11912.15} C_VEL
LIN {X 0,Y 383.013,Z 260.398,A -85,B 0,C 180,E1 -11914.668,E2 -11914.668} C_VEL
LIN {X 0,Y 382.997,Z 260.391,A -85,B 0,C 180,E1 -11917.905,E2 -11917.905} C_VEL
LIN {X 0,Y 382.979,Z 260.397,A -85,B 0,C 180,E1 -11921.348,E2 -11921.348} C_VEL
LIN {X 0,Y 382.992,Z 260.403,A -85,B 0,C 180,E1 -11924.304,E2 -11924.304} C_VEL
LIN {X 0,Y 383.006,Z 260.365,A -85,B 0,C 180,E1 -11927.241,E2 -11927.241} C_VEL
LIN {X 0,Y 383.012,Z 260.39,A -85,B 0,C 180,E1 -11930.414,E2 -11930.414} C_VEL
LIN {X 0,Y 383.022,Z 260.371,A -85,B 0,C 180,E1 -11934.045,E2 -11934.045} C_VEL
LIN {X 0,Y 382.984,Z 260.387,A -85,B 0,C 180,E1 -11937.579,E2 -11937.579} C_VEL
LIN {X 0,Y 383.021,Z 260.631,A -85,B 0,C 180,E1 -11938.162,E2 -11938.162} C_VEL
LIN {X 0,Y 386.546,Z 274.096,A -85,B 0,C 180,E1 -11941.103,E2 -11941.103} C_VEL
LIN {X 0,Y 389.444,Z 287.069,A -85,B 0,C 180,E1 -11943.761,E2 -11943.761} C_VEL
LIN {X 0,Y 389.429,Z 290.173,A -85,B 0,C 180,E1 -11944.334,E2 -11944.334} C_VEL
LIN {X 0,Y 388.546,Z 298.656,A -85,B 0,C 180,E1 -11945.783,E2 -11945.783} C_VEL
LIN {X 0,Y 392.284,Z 323.595,A -85,B 0,C 180,E1 -11946.525,E2 -11946.525} C_VEL
LIN {X 0,Y 390.298,Z 431.191,A -85,B 0,C 180,E1 -11948.615,E2 -11948.615} C_VEL
LIN {X 0,Y 389.6,Z 445.707,A -85,B 0,C 180,E1 -11949.095,E2 -11949.095} C_VEL
LIN {X 0,Y 388.797,Z 459.611,A -85,B 0,C 180,E1 -11949.775,E2 -11949.775} C_VEL
LIN {X 0,Y 387.92,Z 473.192,A -85,B 0,C 180,E1 -11950.673,E2 -11950.673} C_VEL
LIN {X 0,Y 386.826,Z 485.84,A -85,B 0,C 180,E1 -11951.736,E2 -11951.736} C_VEL
LIN {X 0,Y 385.707,Z 497.16,A -85,B 0,C 180,E1 -11952.914,E2 -11952.914} C_VEL
LIN {X 0,Y 384.604,Z 508.466,A -85,B 0,C 180,E1 -11954.364,E2 -11954.364} C_VEL
LIN {X 0,Y 383.705,Z 518.739,A -85,B 0,C 180,E1 -11955.982,E2 -11955.982} C_VEL
LIN {X 0,Y 383.031,Z 526.952,A -85,B 0,C 180,E1 -11957.55,E2 -11957.55} C_VEL
LIN {X 0,Y 382.32,Z 534.922,A -85,B 0,C 180,E1 -11959.408,E2 -11959.408} C_VEL
LIN {X 0,Y 381.986,Z 540.462,A -85,B 0,C 180,E1 -11961.003,E2 -11961.003} C_VEL
LIN {X 0,Y 381.77,Z 544.975,A -85,B 0,C 180,E1 -11962.596,E2 -11962.596} C_VEL
LIN {X 0,Y 381.651,Z 547.996,A -85,B 0,C 180,E1 -11963.931,E2 -11963.931} C_VEL
LIN {X 0,Y 381.603,Z 551.165,A -85,B 0,C 180,E1 -11965.775,E2 -11965.775} C_VEL
LIN {X 0,Y 381.558,Z 553.422,A -85,B 0,C 180,E1 -11967.889,E2 -11967.889} C_VEL
LIN {X 0,Y 381.637,Z 554.253,A -85,B 0,C 180,E1 -11970,E2 -11970} C_VEL
LIN {X 0,Y 381.556,Z 553.661,A -85,B 0,C 180,E1 -11972.111,E2 -11972.111} C_VEL
LIN {X 0,Y 381.606,Z 551.624,A -85,B 0,C 180,E1 -11974.225,E2 -11974.225} C_VEL
LIN {X 0,Y 381.7,Z 548.107,A -85,B 0,C 180,E1 -11976.343,E2 -11976.343} C_VEL
LIN {X 0,Y 381.94,Z 543.024,A -85,B 0,C 180,E1 -11978.465,E2 -11978.465} C_VEL
LIN {X 0,Y 382.275,Z 538.086,A -85,B 0,C 180,E1 -11980.058,E2 -11980.058} C_VEL
LIN {X 0,Y 382.909,Z 530.935,A -85,B 0,C 180,E1 -11981.916,E2 -11981.916} C_VEL
LIN {X 0,Y 383.735,Z 522.049,A -85,B 0,C 180,E1 -11983.774,E2 -11983.774} C_VEL
LIN {X 0,Y 384.642,Z 512.725,A -85,B 0,C 180,E1 -11985.363,E2 -11985.363} C_VEL
LIN {X 0,Y 385.711,Z 502.385,A -85,B 0,C 180,E1 -11986.813,E2 -11986.813} C_VEL
LIN {X 0,Y 386.941,Z 490.935,A -85,B 0,C 180,E1 -11988.122,E2 -11988.122} C_VEL
LIN {X 0,Y 388.111,Z 479.095,A -85,B 0,C 180,E1 -11989.223,E2 -11989.223} C_VEL
LIN {X 0,Y 388.995,Z 467.85,A -85,B 0,C 180,E1 -11990.076,E2 -11990.076} C_VEL
LIN {X 0,Y 389.943,Z 454.727,A -85,B 0,C 180,E1 -11990.852,E2 -11990.852} C_VEL
LIN {X 0,Y 390.767,Z 440.543,A -85,B 0,C 180,E1 -11991.462,E2 -11991.462} C_VEL
LIN {X 0,Y 391.319,Z 426.895,A -85,B 0,C 180,E1 -11991.845,E2 -11991.845} C_VEL
LIN {X 0,Y 393.292,Z 323.391,A -85,B 0,C 180,E1 -11993.851,E2 -11993.851} C_VEL
LIN {X 0,Y 389.213,Z 298.49,A -85,B 0,C 180,E1 -11994.657,E2 -11994.657} C_VEL
LIN {X 0,Y 390.184,Z 289.769,A -85,B 0,C 180,E1 -11996.185,E2 -11996.185} C_VEL
LIN {X 0,Y 388.287,Z 280.608,A -85,B 0,C 180,E1 -11998.073,E2 -11998.073} C_VEL
LIN {X 0,Y 384.952,Z 267.63,A -85,B 0,C 180,E1 -12000.899,E2 -12000.899} C_VEL
LIN {X 0,Y 383.013,Z 260.463,A -85,B 0,C 180,E1 -12002.594,E2 -12002.594} C_VEL
LIN {X 0,Y 383.029,Z 260.366,A -85,B 0,C 180,E1 -12006.164,E2 -12006.164} C_VEL
LIN {X 0,Y 383.012,Z 260.397,A -85,B 0,C 180,E1 -12009.957,E2 -12009.957} C_VEL
LIN {X 0,Y 383.062,Z 260.394,A -85,B 0,C 180,E1 -12012.788,E2 -12012.788} C_VEL
LIN {X 0,Y 383.004,Z 260.398,A -85,B 0,C 180,E1 -12015.79,E2 -12015.79} C_VEL
LIN {X 0,Y 382.984,Z 260.389,A -85,B 0,C 180,E1 -12018.795,E2 -12018.795} C_VEL
LIN {X 0,Y 382.997,Z 260.399,A -85,B 0,C 180,E1 -12022.096,E2 -12022.096} C_VEL
LIN {X 0,Y 383.013,Z 260.391,A -85,B 0,C 180,E1 -12025.332,E2 -12025.332} C_VEL
LIN {X 0,Y 382.981,Z 260.39,A -85,B 0,C 180,E1 -12029.082,E2 -12029.082} C_VEL
LIN {X 0,Y 383.051,Z 260.393,A -85,B 0,C 180,E1 -12032.698,E2 -12032.698} C_VEL
LIN {X 0,Y 383.028,Z 260.396,A -85,B 0,C 180,E1 -12036.193,E2 -12036.193} C_VEL
LIN {X 0,Y 383.049,Z 260.39,A -85,B 0,C 180,E1 -12039.598,E2 -12039.598} C_VEL
LIN {X 0,Y 383.099,Z 260.384,A -85,B 0,C 180,E1 -12042.931,E2 -12042.931} C_VEL
LIN {X 0,Y 383.119,Z 260.384,A -85,B 0,C 180,E1 -12046.464,E2 -12046.464} C_VEL
LIN {X 0,Y 383.145,Z 260.381,A -85,B 0,C 180,E1 -12050.498,E2 -12050.498} C_VEL
LIN {X 0,Y 383.277,Z 260.362,A -85,B 0,C 180,E1 -12053.684,E2 -12053.684} C_VEL
LIN {X 0,Y 383.382,Z 260.348,A -85,B 0,C 180,E1 -12057.899,E2 -12057.899} C_VEL
LIN {X 0,Y 383.513,Z 260.337,A -85,B 0,C 180,E1 -12060,E2 -12060} C_VEL
LIN {X 0,Y 383.246,Z 260.364,A -85,B 0,C 180,E1 -12063.154,E2 -12063.154} C_VEL
LIN {X 0,Y 383.263,Z 260.36,A -85,B 0,C 180,E1 -12066.642,E2 -12066.642} C_VEL
LIN {X 0,Y 383.255,Z 260.366,A -85,B 0,C 180,E1 -12068.436,E2 -12068.436} C_VEL
LIN {X 0,Y 383.092,Z 260.384,A -85,B 0,C 180,E1 -12071.643,E2 -12071.643} C_VEL
LIN {X 0,Y 383.105,Z 260.388,A -85,B 0,C 180,E1 -12074.882,E2 -12074.882} C_VEL
LIN {X 0,Y 383.058,Z 260.393,A -85,B 0,C 180,E1 -12078.174,E2 -12078.174} C_VEL
LIN {X 0,Y 382.995,Z 260.404,A -85,B 0,C 180,E1 -12081.531,E2 -12081.531} C_VEL
LIN {X 0,Y 383.048,Z 260.395,A -85,B 0,C 180,E1 -12084.961,E2 -12084.961} C_VEL
LIN {X 0,Y 383.026,Z 260.382,A -85,B 0,C 180,E1 -12088.271,E2 -12088.271} C_VEL
LIN {X 0,Y 383.007,Z 260.401,A -85,B 0,C 180,E1 -12092.151,E2 -12092.151} C_VEL
LIN {X 0,Y 383.016,Z 260.384,A -85,B 0,C 180,E1 -12094.669,E2 -12094.669} C_VEL
LIN {X 0,Y 382.999,Z 260.401,A -85,B 0,C 180,E1 -12097.905,E2 -12097.905} C_VEL
LIN {X 0,Y 382.983,Z 260.401,A -85,B 0,C 180,E1 -12101.348,E2 -12101.348} C_VEL
LIN {X 0,Y 382.996,Z 260.392,A -85,B 0,C 180,E1 -12104.304,E2 -12104.304} C_VEL
LIN {X 0,Y 383.01,Z 260.393,A -85,B 0,C 180,E1 -12107.241,E2 -12107.241} C_VEL
LIN {X 0,Y 383.016,Z 260.382,A -85,B 0,C 180,E1 -12110.414,E2 -12110.414} C_VEL
LIN {X 0,Y 383.026,Z 260.402,A -85,B 0,C 180,E1 -12114.045,E2 -12114.045} C_VEL
LIN {X 0,Y 383.091,Z 260.612,A -85,B 0,C 180,E1 -12115.06,E2 -12115.06} C_VEL
LIN {X 0,Y 386.263,Z 273.266,A -85,B 0,C 180,E1 -12118.154,E2 -12118.154} C_VEL
LIN {X 0,Y 389.095,Z 286.107,A -85,B 0,C 180,E1 -12121.108,E2 -12121.108} C_VEL
LIN {X 0,Y 389.229,Z 288.945,A -85,B 0,C 180,E1 -12121.708,E2 -12121.708} C_VEL
LIN {X 0,Y 387.326,Z 307.345,A -85,B 0,C 180,E1 -12125.334,E2 -12125.334} C_VEL
LIN {X 0,Y 386.924,Z 312.511,A -85,B 0,C 180,E1 -12126.274,E2 -12126.274} C_VEL
LIN {X 0,Y 392.419,Z 341.958,A -85,B 0,C 180,E1 -12127.188,E2 -12127.188} C_VEL
LIN {X 0,Y 391.306,Z 424.621,A -85,B 0,C 180,E1 -12128.638,E2 -12128.638} C_VEL
LIN {X 0,Y 390.71,Z 438.067,A -85,B 0,C 180,E1 -12129.045,E2 -12129.045} C_VEL
LIN {X 0,Y 390.151,Z 450.504,A -85,B 0,C 180,E1 -12129.645,E2 -12129.645} C_VEL
LIN {X 0,Y 389.135,Z 463.326,A -85,B 0,C 180,E1 -12130.481,E2 -12130.481} C_VEL
LIN {X 0,Y 388.142,Z 474.005,A -85,B 0,C 180,E1 -12131.39,E2 -12131.39} C_VEL
LIN {X 0,Y 386.898,Z 484.945,A -85,B 0,C 180,E1 -12132.559,E2 -12132.559} C_VEL
LIN {X 0,Y 385.74,Z 494.731,A -85,B 0,C 180,E1 -12133.868,E2 -12133.868} C_VEL
LIN {X 0,Y 384.558,Z 504.237,A -85,B 0,C 180,E1 -12135.447,E2 -12135.447} C_VEL
LIN {X 0,Y 383.773,Z 511.856,A -85,B 0,C 180,E1 -12137.037,E2 -12137.037} C_VEL
LIN {X 0,Y 382.836,Z 518.871,A -85,B 0,C 180,E1 -12138.886,E2 -12138.886} C_VEL
LIN {X 0,Y 382.361,Z 523.587,A -85,B 0,C 180,E1 -12140.478,E2 -12140.478} C_VEL
LIN {X 0,Y 382.043,Z 527.245,A -85,B 0,C 180,E1 -12142.07,E2 -12142.07} C_VEL
LIN {X 0,Y 381.764,Z 530.105,A -85,B 0,C 180,E1 -12143.779,E2 -12143.779} C_VEL
LIN {X 0,Y 381.643,Z 532.145,A -85,B 0,C 180,E1 -12145.776,E2 -12145.776} C_VEL
LIN {X 0,Y 381.613,Z 532.883,A -85,B 0,C 180,E1 -12147.889,E2 -12147.889} C_VEL
LIN {X 0,Y 381.643,Z 532.111,A -85,B 0,C 180,E1 -12150,E2 -12150} C_VEL
LIN {X 0,Y 381.799,Z 529.888,A -85,B 0,C 180,E1 -12152.11,E2 -12152.11} C_VEL
LIN {X 0,Y 382.064,Z 527.172,A -85,B 0,C 180,E1 -12153.691,E2 -12153.691} C_VEL
LIN {X 0,Y 382.224,Z 523.515,A -85,B 0,C 180,E1 -12155.275,E2 -12155.275} C_VEL
LIN {X 0,Y 382.724,Z 518.797,A -85,B 0,C 180,E1 -12156.855,E2 -12156.855} C_VEL
LIN {X 0,Y 383.417,Z 511.803,A -85,B 0,C 180,E1 -12158.698,E2 -12158.698} C_VEL
LIN {X 0,Y 383.925,Z 506.76,A -85,B 0,C 180,E1 -12159.777,E2 -12159.777} C_VEL
LIN {X 0,Y 383.701,Z 503.215,A -85,B 0,C 180,E1 -12160.479,E2 -12160.479} C_VEL
LIN {X 0,Y 381.65,Z 497.159,A -85,B 0,C 180,E1 -12161.615,E2 -12161.615} C_VEL
LIN {X 0,Y 379.581,Z 490.612,A -85,B 0,C 180,E1 -12162.692,E2 -12162.692} C_VEL
LIN {X 0,Y 379.324,Z 486.234,A -85,B 0,C 180,E1 -12163.295,E2 -12163.295} C_VEL
LIN {X 0,Y 380.413,Z 476.041,A -85,B 0,C 180,E1 -12164.442,E2 -12164.442} C_VEL
LIN {X 0,Y 381.119,Z 467.503,A -85,B 0,C 180,E1 -12165.234,E2 -12165.234} C_VEL
LIN {X 0,Y 382.015,Z 457.052,A -85,B 0,C 180,E1 -12166.019,E2 -12166.019} C_VEL
LIN {X 0,Y 382.908,Z 444.505,A -85,B 0,C 180,E1 -12166.734,E2 -12166.734} C_VEL
LIN {X 0,Y 383.489,Z 431.48,A -85,B 0,C 180,E1 -12167.254,E2 -12167.254} C_VEL
LIN {X 0,Y 383.833,Z 417.067,A -85,B 0,C 180,E1 -12167.584,E2 -12167.584} C_VEL
LIN {X 0,Y 384.781,Z 342.436,A -85,B 0,C 180,E1 -12168.899,E2 -12168.899} C_VEL
LIN {X 0,Y 379.625,Z 312.395,A -85,B 0,C 180,E1 -12169.792,E2 -12169.792} C_VEL
LIN {X 0,Y 379.91,Z 308.058,A -85,B 0,C 180,E1 -12170.578,E2 -12170.578} C_VEL
LIN {X 0,Y 381.816,Z 288.537,A -85,B 0,C 180,E1 -12174.465,E2 -12174.465} C_VEL
LIN {X 0,Y 381.6,Z 285.761,A -85,B 0,C 180,E1 -12175.061,E2 -12175.061} C_VEL
LIN {X 0,Y 378.635,Z 271.891,A -85,B 0,C 180,E1 -12178.249,E2 -12178.249} C_VEL
LIN {X 0,Y 375.966,Z 261.394,A -85,B 0,C 180,E1 -12180.832,E2 -12180.832} C_VEL
LIN {X 0,Y 375.981,Z 261.257,A -85,B 0,C 180,E1 -12184.666,E2 -12184.666} C_VEL
LIN {X 0,Y 375.975,Z 261.272,A -85,B 0,C 180,E1 -12188.27,E2 -12188.27} C_VEL
LIN {X 0,Y 375.935,Z 261.275,A -85,B 0,C 180,E1 -12191.6,E2 -12191.6} C_VEL
LIN {X 0,Y 375.927,Z 261.271,A -85,B 0,C 180,E1 -12195.268,E2 -12195.268} C_VEL
LIN {X 0,Y 375.933,Z 261.28,A -85,B 0,C 180,E1 -12198.398,E2 -12198.398} C_VEL
LIN {X 0,Y 375.972,Z 261.274,A -85,B 0,C 180,E1 -12201.729,E2 -12201.729} C_VEL
LIN {X 0,Y 375.977,Z 261.258,A -85,B 0,C 180,E1 -12205.332,E2 -12205.332} C_VEL
LIN {X 0,Y 375.957,Z 261.272,A -85,B 0,C 180,E1 -12208.437,E2 -12208.437} C_VEL
LIN {X 0,Y 375.999,Z 261.266,A -85,B 0,C 180,E1 -12212.141,E2 -12212.141} C_VEL
LIN {X 0,Y 376.002,Z 261.275,A -85,B 0,C 180,E1 -12214.538,E2 -12214.538} C_VEL
LIN {X 0,Y 375.958,Z 261.277,A -85,B 0,C 180,E1 -12218.045,E2 -12218.045} C_VEL
LIN {X 0,Y 376.004,Z 261.27,A -85,B 0,C 180,E1 -12221.472,E2 -12221.472} C_VEL
LIN {X 0,Y 376.054,Z 261.259,A -85,B 0,C 180,E1 -12224.832,E2 -12224.832} C_VEL
LIN {X 0,Y 376.044,Z 261.268,A -85,B 0,C 180,E1 -12228.136,E2 -12228.136} C_VEL
LIN {X 0,Y 376.214,Z 261.244,A -85,B 0,C 180,E1 -12231.918,E2 -12231.918} C_VEL
LIN {X 0,Y 376.165,Z 261.245,A -85,B 0,C 180,E1 -12234.639,E2 -12234.639} C_VEL
LIN {X 0,Y 376.348,Z 261.229,A -85,B 0,C 180,E1 -12237.859,E2 -12237.859} C_VEL
LIN {X 0,Y 376.482,Z 261.208,A -85,B 0,C 180,E1 -12240,E2 -12240} C_VEL
LIN {X 0,Y 376.184,Z 261.249,A -85,B 0,C 180,E1 -12243.213,E2 -12243.213} C_VEL
LIN {X 0,Y 376.24,Z 261.236,A -85,B 0,C 180,E1 -12246.435,E2 -12246.435} C_VEL
LIN {X 0,Y 376.199,Z 261.249,A -85,B 0,C 180,E1 -12248.595,E2 -12248.595} C_VEL
LIN {X 0,Y 376.042,Z 261.26,A -85,B 0,C 180,E1 -12251.863,E2 -12251.863} C_VEL
LIN {X 0,Y 376.052,Z 261.261,A -85,B 0,C 180,E1 -12255.167,E2 -12255.167} C_VEL
LIN {X 0,Y 376.017,Z 261.271,A -85,B 0,C 180,E1 -12258.526,E2 -12258.526} C_VEL
LIN {X 0,Y 375.957,Z 261.277,A -85,B 0,C 180,E1 -12261.954,E2 -12261.954} C_VEL
LIN {X 0,Y 376,Z 261.267,A -85,B 0,C 180,E1 -12265.461,E2 -12265.461} C_VEL
LIN {X 0,Y 375.971,Z 261.266,A -85,B 0,C 180,E1 -12269.079,E2 -12269.079} C_VEL
LIN {X 0,Y 375.946,Z 261.278,A -85,B 0,C 180,E1 -12272.829,E2 -12272.829} C_VEL
LIN {X 0,Y 375.953,Z 261.273,A -85,B 0,C 180,E1 -12275.416,E2 -12275.416} C_VEL
LIN {X 0,Y 375.971,Z 261.272,A -85,B 0,C 180,E1 -12278.271,E2 -12278.271} C_VEL
LIN {X 0,Y 375.93,Z 261.272,A -85,B 0,C 180,E1 -12281.601,E2 -12281.601} C_VEL
LIN {X 0,Y 375.949,Z 261.277,A -85,B 0,C 180,E1 -12285.265,E2 -12285.265} C_VEL
LIN {X 0,Y 375.936,Z 261.244,A -85,B 0,C 180,E1 -12289.133,E2 -12289.133} C_VEL
LIN {X 0,Y 375.962,Z 261.277,A -85,B 0,C 180,E1 -12291.912,E2 -12291.912} C_VEL
LIN {X 0,Y 375.977,Z 261.257,A -85,B 0,C 180,E1 -12295.333,E2 -12295.333} C_VEL
LIN {X 0,Y 375.976,Z 261.459,A -85,B 0,C 180,E1 -12297.676,E2 -12297.676} C_VEL
LIN {X 0,Y 379.624,Z 275.452,A -85,B 0,C 180,E1 -12300.809,E2 -12300.809} C_VEL
LIN {X 0,Y 382.563,Z 288.516,A -85,B 0,C 180,E1 -12303.546,E2 -12303.546} C_VEL
LIN {X 0,Y 382.771,Z 290.072,A -85,B 0,C 180,E1 -12303.855,E2 -12303.855} C_VEL
LIN {X 0,Y 381.819,Z 298.672,A -85,B 0,C 180,E1 -12305.37,E2 -12305.37} C_VEL
LIN {X 0,Y 385.684,Z 324.626,A -85,B 0,C 180,E1 -12306.163,E2 -12306.163} C_VEL
LIN {X 0,Y 383.614,Z 430.918,A -85,B 0,C 180,E1 -12308.259,E2 -12308.259} C_VEL
LIN {X 0,Y 382.917,Z 445.524,A -85,B 0,C 180,E1 -12308.747,E2 -12308.747} C_VEL
LIN {X 0,Y 382.026,Z 460.017,A -85,B 0,C 180,E1 -12309.471,E2 -12309.471} C_VEL
LIN {X 0,Y 381.134,Z 473.223,A -85,B 0,C 180,E1 -12310.364,E2 -12310.364} C_VEL
LIN {X 0,Y 380.032,Z 485.339,A -85,B 0,C 180,E1 -12311.398,E2 -12311.398} C_VEL
LIN {X 0,Y 378.863,Z 496.726,A -85,B 0,C 180,E1 -12312.595,E2 -12312.595} C_VEL
LIN {X 0,Y 377.699,Z 508.099,A -85,B 0,C 180,E1 -12314.071,E2 -12314.071} C_VEL
LIN {X 0,Y 376.792,Z 518.254,A -85,B 0,C 180,E1 -12315.692,E2 -12315.692} C_VEL
LIN {X 0,Y 376.02,Z 526.647,A -85,B 0,C 180,E1 -12317.314,E2 -12317.314} C_VEL
LIN {X 0,Y 375.295,Z 534.641,A -85,B 0,C 180,E1 -12319.207,E2 -12319.207} C_VEL
LIN {X 0,Y 374.92,Z 540.2,A -85,B 0,C 180,E1 -12320.832,E2 -12320.832} C_VEL
LIN {X 0,Y 374.687,Z 544.73,A -85,B 0,C 180,E1 -12322.456,E2 -12322.456} C_VEL
LIN {X 0,Y 374.544,Z 548.108,A -85,B 0,C 180,E1 -12323.987,E2 -12323.987} C_VEL
LIN {X 0,Y 374.505,Z 550.942,A -85,B 0,C 180,E1 -12325.695,E2 -12325.695} C_VEL
LIN {X 0,Y 374.457,Z 553.21,A -85,B 0,C 180,E1 -12327.849,E2 -12327.849} C_VEL
LIN {X 0,Y 374.552,Z 554.052,A -85,B 0,C 180,E1 -12330,E2 -12330} C_VEL
LIN {X 0,Y 374.455,Z 553.469,A -85,B 0,C 180,E1 -12332.151,E2 -12332.151} C_VEL
LIN {X 0,Y 374.509,Z 551.442,A -85,B 0,C 180,E1 -12334.305,E2 -12334.305} C_VEL
LIN {X 0,Y 374.62,Z 547.931,A -85,B 0,C 180,E1 -12336.463,E2 -12336.463} C_VEL
LIN {X 0,Y 374.867,Z 542.852,A -85,B 0,C 180,E1 -12338.626,E2 -12338.626} C_VEL
LIN {X 0,Y 375.219,Z 537.919,A -85,B 0,C 180,E1 -12340.25,E2 -12340.25} C_VEL
LIN {X 0,Y 375.918,Z 530.771,A -85,B 0,C 180,E1 -12342.141,E2 -12342.141} C_VEL
LIN {X 0,Y 376.788,Z 521.887,A -85,B 0,C 180,E1 -12344.033,E2 -12344.033} C_VEL
LIN {X 0,Y 377.747,Z 512.564,A -85,B 0,C 180,E1 -12345.651,E2 -12345.651} C_VEL
LIN {X 0,Y 378.882,Z 502.223,A -85,B 0,C 180,E1 -12347.126,E2 -12347.126} C_VEL
LIN {X 0,Y 380.158,Z 490.766,A -85,B 0,C 180,E1 -12348.457,E2 -12348.457} C_VEL
LIN {X 0,Y 381.446,Z 478.157,A -85,B 0,C 180,E1 -12349.639,E2 -12349.639} C_VEL
LIN {X 0,Y 382.502,Z 465.667,A -85,B 0,C 180,E1 -12350.572,E2 -12350.572} C_VEL
LIN {X 0,Y 383.475,Z 451.918,A -85,B 0,C 180,E1 -12351.361,E2 -12351.361} C_VEL
LIN {X 0,Y 384.346,Z 437.526,A -85,B 0,C 180,E1 -12351.944,E2 -12351.944} C_VEL
LIN {X 0,Y 384.814,Z 423.356,A -85,B 0,C 180,E1 -12352.305,E2 -12352.305} C_VEL
LIN {X 0,Y 386.771,Z 324.185,A -85,B 0,C 180,E1 -12354.251,E2 -12354.251} C_VEL
LIN {X 0,Y 382.575,Z 298.676,A -85,B 0,C 180,E1 -12355.096,E2 -12355.096} C_VEL
LIN {X 0,Y 383.383,Z 291.391,A -85,B 0,C 180,E1 -12356.393,E2 -12356.393} C_VEL
LIN {X 0,Y 381.338,Z 281.83,A -85,B 0,C 180,E1 -12358.41,E2 -12358.41} C_VEL
LIN {X 0,Y 378.087,Z 269.16,A -85,B 0,C 180,E1 -12361.234,E2 -12361.234} C_VEL
LIN {X 0,Y 375.978,Z 261.363,A -85,B 0,C 180,E1 -12363.104,E2 -12363.104} C_VEL
LIN {X 0,Y 375.961,Z 261.245,A -85,B 0,C 180,E1 -12366.504,E2 -12366.504} C_VEL
LIN {X 0,Y 375.991,Z 261.271,A -85,B 0,C 180,E1 -12369.971,E2 -12369.971} C_VEL
LIN {X 0,Y 375.987,Z 261.274,A -85,B 0,C 180,E1 -12373.198,E2 -12373.198} C_VEL
LIN {X 0,Y 375.933,Z 261.281,A -85,B 0,C 180,E1 -12376.81,E2 -12376.81} C_VEL
LIN {X 0,Y 375.96,Z 261.279,A -85,B 0,C 180,E1 -12380.537,E2 -12380.537} C_VEL
LIN {X 0,Y 375.96,Z 261.262,A -85,B 0,C 180,E1 -12383.495,E2 -12383.495} C_VEL
LIN {X 0,Y 375.955,Z 261.274,A -85,B 0,C 180,E1 -12385.888,E2 -12385.888} C_VEL
LIN {X 0,Y 375.963,Z 261.256,A -85,B 0,C 180,E1 -12389.688,E2 -12389.688} C_VEL
LIN {X 0,Y 375.997,Z 261.266,A -85,B 0,C 180,E1 -12392.142,E2 -12392.142} C_VEL
LIN {X 0,Y 376.001,Z 261.27,A -85,B 0,C 180,E1 -12394.539,E2 -12394.539} C_VEL
LIN {X 0,Y 375.958,Z 261.278,A -85,B 0,C 180,E1 -12398.046,E2 -12398.046} C_VEL
LIN {X 0,Y 376.018,Z 261.271,A -85,B 0,C 180,E1 -12401.474,E2 -12401.474} C_VEL
LIN {X 0,Y 376.052,Z 261.262,A -85,B 0,C 180,E1 -12404.833,E2 -12404.833} C_VEL
LIN {X 0,Y 376.043,Z 261.26,A -85,B 0,C 180,E1 -12408.137,E2 -12408.137} C_VEL
LIN {X 0,Y 376.213,Z 261.239,A -85,B 0,C 180,E1 -12411.919,E2 -12411.919} C_VEL
LIN {X 0,Y 376.165,Z 261.251,A -85,B 0,C 180,E1 -12414.64,E2 -12414.64} C_VEL
LIN {X 0,Y 376.348,Z 261.224,A -85,B 0,C 180,E1 -12417.86,E2 -12417.86} C_VEL
LIN {X 0,Y 376.483,Z 261.213,A -85,B 0,C 180,E1 -12420,E2 -12420} C_VEL
LIN {X 0,Y 376.184,Z 261.244,A -85,B 0,C 180,E1 -12423.213,E2 -12423.213} C_VEL
LIN {X 0,Y 376.228,Z 261.236,A -85,B 0,C 180,E1 -12426.634,E2 -12426.634} C_VEL
LIN {X 0,Y 376.2,Z 261.245,A -85,B 0,C 180,E1 -12428.596,E2 -12428.596} C_VEL
LIN {X 0,Y 376.044,Z 261.262,A -85,B 0,C 180,E1 -12431.864,E2 -12431.864} C_VEL
LIN {X 0,Y 376.054,Z 261.263,A -85,B 0,C 180,E1 -12435.168,E2 -12435.168} C_VEL
LIN {X 0,Y 376.005,Z 261.272,A -85,B 0,C 180,E1 -12438.527,E2 -12438.527} C_VEL
LIN {X 0,Y 375.964,Z 261.277,A -85,B 0,C 180,E1 -12441.955,E2 -12441.955} C_VEL
LIN {X 0,Y 376.003,Z 261.275,A -85,B 0,C 180,E1 -12445.462,E2 -12445.462} C_VEL
LIN {X 0,Y 375.957,Z 261.257,A -85,B 0,C 180,E1 -12449.081,E2 -12449.081} C_VEL
LIN {X 0,Y 375.947,Z 261.281,A -85,B 0,C 180,E1 -12452.829,E2 -12452.829} C_VEL
LIN {X 0,Y 375.956,Z 261.263,A -85,B 0,C 180,E1 -12455.416,E2 -12455.416} C_VEL
LIN {X 0,Y 375.973,Z 261.277,A -85,B 0,C 180,E1 -12458.271,E2 -12458.271} C_VEL
LIN {X 0,Y 375.933,Z 261.282,A -85,B 0,C 180,E1 -12461.602,E2 -12461.602} C_VEL
LIN {X 0,Y 375.928,Z 261.281,A -85,B 0,C 180,E1 -12465.269,E2 -12465.269} C_VEL
LIN {X 0,Y 375.936,Z 261.277,A -85,B 0,C 180,E1 -12468.4,E2 -12468.4} C_VEL
LIN {X 0,Y 375.975,Z 261.245,A -85,B 0,C 180,E1 -12471.73,E2 -12471.73} C_VEL
LIN {X 0,Y 376.032,Z 261.44,A -85,B 0,C 180,E1 -12474.532,E2 -12474.532} C_VEL
LIN {X 0,Y 379.256,Z 274.257,A -85,B 0,C 180,E1 -12477.746,E2 -12477.746} C_VEL
LIN {X 0,Y 381.886,Z 285.968,A -85,B 0,C 180,E1 -12480.509,E2 -12480.509} C_VEL
LIN {X 0,Y 382.459,Z 290.237,A -85,B 0,C 180,E1 -12481.461,E2 -12481.461} C_VEL
LIN {X 0,Y 380.618,Z 307.241,A -85,B 0,C 180,E1 -12484.869,E2 -12484.869} C_VEL
LIN {X 0,Y 380.2,Z 312.39,A -85,B 0,C 180,E1 -12485.821,E2 -12485.821} C_VEL
LIN {X 0,Y 385.765,Z 341.847,A -85,B 0,C 180,E1 -12486.766,E2 -12486.766} C_VEL
LIN {X 0,Y 385.949,Z 346.6,A -85,B 0,C 180,E1 -12486.866,E2 -12486.866} C_VEL
LIN {X 0,Y 384.676,Z 426.228,A -85,B 0,C 180,E1 -12488.287,E2 -12488.287} C_VEL
LIN {X 0,Y 384.044,Z 439.583,A -85,B 0,C 180,E1 -12488.728,E2 -12488.728} C_VEL
LIN {X 0,Y 383.36,Z 452.556,A -85,B 0,C 180,E1 -12489.388,E2 -12489.388} C_VEL
LIN {X 0,Y 382.293,Z 465.13,A -85,B 0,C 180,E1 -12490.257,E2 -12490.257} C_VEL
LIN {X 0,Y 381.085,Z 476.732,A -85,B 0,C 180,E1 -12491.311,E2 -12491.311} C_VEL
LIN {X 0,Y 379.868,Z 487.17,A -85,B 0,C 180,E1 -12492.504,E2 -12492.504} C_VEL
LIN {X 0,Y 378.666,Z 496.604,A -85,B 0,C 180,E1 -12493.836,E2 -12493.836} C_VEL
LIN {X 0,Y 377.629,Z 504.627,A -85,B 0,C 180,E1 -12495.224,E2 -12495.224} C_VEL
LIN {X 0,Y 376.833,Z 511.99,A -85,B 0,C 180,E1 -12496.793,E2 -12496.793} C_VEL
LIN {X 0,Y 376.083,Z 517.195,A -85,B 0,C 180,E1 -12498.138,E2 -12498.138} C_VEL
LIN {X 0,Y 375.478,Z 522.302,A -85,B 0,C 180,E1 -12499.758,E2 -12499.758} C_VEL
LIN {X 0,Y 375.095,Z 526.302,A -85,B 0,C 180,E1 -12501.379,E2 -12501.379} C_VEL
LIN {X 0,Y 374.884,Z 528.436,A -85,B 0,C 180,E1 -12502.459,E2 -12502.459} C_VEL
LIN {X 0,Y 374.619,Z 531.409,A -85,B 0,C 180,E1 -12504.618,E2 -12504.618} C_VEL
LIN {X 0,Y 374.495,Z 532.888,A -85,B 0,C 180,E1 -12506.773,E2 -12506.773} C_VEL
LIN {X 0,Y 374.512,Z 533.083,A -85,B 0,C 180,E1 -12507.849,E2 -12507.849} C_VEL
LIN {X 0,Y 374.559,Z 532.326,A -85,B 0,C 180,E1 -12510,E2 -12510} C_VEL
LIN {X 0,Y 374.707,Z 530.118,A -85,B 0,C 180,E1 -12512.15,E2 -12512.15} C_VEL
LIN {X 0,Y 374.988,Z 527.419,A -85,B 0,C 180,E1 -12513.761,E2 -12513.761} C_VEL
LIN {X 0,Y 375.175,Z 523.78,A -85,B 0,C 180,E1 -12515.374,E2 -12515.374} C_VEL
LIN {X 0,Y 375.682,Z 519.085,A -85,B 0,C 180,E1 -12516.984,E2 -12516.984} C_VEL
LIN {X 0,Y 376.403,Z 512.116,A -85,B 0,C 180,E1 -12518.861,E2 -12518.861} C_VEL
LIN {X 0,Y 377.264,Z 504.571,A -85,B 0,C 180,E1 -12520.465,E2 -12520.465} C_VEL
LIN {X 0,Y 378.367,Z 495.16,A -85,B 0,C 180,E1 -12522.061,E2 -12522.061} C_VEL
LIN {X 0,Y 379.324,Z 486.234,A -85,B 0,C 180,E1 -12523.295,E2 -12523.295} C_VEL
LIN {X 0,Y 378.91,Z 483.255,A -85,B 0,C 180,E1 -12523.693,E2 -12523.693} C_VEL
LIN {X 0,Y 374.316,Z 473.752,A -85,B 0,C 180,E1 -12524.975,E2 -12524.975} C_VEL
LIN {X 0,Y 374.072,Z 470.432,A -85,B 0,C 180,E1 -12525.315,E2 -12525.315} C_VEL
LIN {X 0,Y 375.151,Z 459.722,A -85,B 0,C 180,E1 -12526.18,E2 -12526.18} C_VEL
LIN {X 0,Y 375.997,Z 448.06,A -85,B 0,C 180,E1 -12526.911,E2 -12526.911} C_VEL
LIN {X 0,Y 376.664,Z 434.635,A -85,B 0,C 180,E1 -12527.509,E2 -12527.509} C_VEL
LIN {X 0,Y 377.119,Z 421.107,A -85,B 0,C 180,E1 -12527.879,E2 -12527.879} C_VEL
LIN {X 0,Y 378.19,Z 343.644,A -85,B 0,C 180,E1 -12529.267,E2 -12529.267} C_VEL
LIN {X 0,Y 373.008,Z 313.408,A -85,B 0,C 180,E1 -12530.169,E2 -12530.169} C_VEL
LIN {X 0,Y 372.8,Z 311.728,A -85,B 0,C 180,E1 -12530.282,E2 -12530.282} C_VEL
LIN {X 0,Y 374.5,Z 294.223,A -85,B 0,C 180,E1 -12533.795,E2 -12533.795} C_VEL
LIN {X 0,Y 374.98,Z 288.652,A -85,B 0,C 180,E1 -12534.942,E2 -12534.942} C_VEL
LIN {X 0,Y 372.077,Z 274.774,A -85,B 0,C 180,E1 -12538.177,E2 -12538.177} C_VEL
LIN {X 0,Y 368.937,Z 262.353,A -85,B 0,C 180,E1 -12541.27,E2 -12541.27} C_VEL
LIN {X 0,Y 368.93,Z 262.139,A -85,B 0,C 180,E1 -12545.001,E2 -12545.001} C_VEL
LIN {X 0,Y 368.909,Z 262.154,A -85,B 0,C 180,E1 -12548.639,E2 -12548.639} C_VEL
LIN {X 0,Y 368.882,Z 262.157,A -85,B 0,C 180,E1 -12552.009,E2 -12552.009} C_VEL
LIN {X 0,Y 368.88,Z 262.148,A -85,B 0,C 180,E1 -12555.175,E2 -12555.175} C_VEL
LIN {X 0,Y 368.881,Z 262.159,A -85,B 0,C 180,E1 -12558.177,E2 -12558.177} C_VEL
LIN {X 0,Y 368.906,Z 262.146,A -85,B 0,C 180,E1 -12561.359,E2 -12561.359} C_VEL
LIN {X 0,Y 368.934,Z 262.136,A -85,B 0,C 180,E1 -12565.146,E2 -12565.146} C_VEL
LIN {X 0,Y 368.926,Z 262.154,A -85,B 0,C 180,E1 -12569.046,E2 -12569.046} C_VEL
LIN {X 0,Y 368.983,Z 262.14,A -85,B 0,C 180,E1 -12571.564,E2 -12571.564} C_VEL
LIN {X 0,Y 368.996,Z 262.145,A -85,B 0,C 180,E1 -12574.019,E2 -12574.019} C_VEL
LIN {X 0,Y 368.923,Z 262.154,A -85,B 0,C 180,E1 -12577.604,E2 -12577.604} C_VEL
LIN {X 0,Y 368.953,Z 262.148,A -85,B 0,C 180,E1 -12581.105,E2 -12581.105} C_VEL
LIN {X 0,Y 368.993,Z 262.14,A -85,B 0,C 180,E1 -12584.535,E2 -12584.535} C_VEL
LIN {X 0,Y 369,Z 262.144,A -85,B 0,C 180,E1 -12587.906,E2 -12587.906} C_VEL
LIN {X 0,Y 369.161,Z 262.122,A -85,B 0,C 180,E1 -12591.868,E2 -12591.868} C_VEL
LIN {X 0,Y 369.137,Z 262.121,A -85,B 0,C 180,E1 -12594.537,E2 -12594.537} C_VEL
LIN {X 0,Y 369.313,Z 262.105,A -85,B 0,C 180,E1 -12597.818,E2 -12597.818} C_VEL
LIN {X 0,Y 369.452,Z 262.084,A -85,B 0,C 180,E1 -12600,E2 -12600} C_VEL
LIN {X 0,Y 369.312,Z 262.102,A -85,B 0,C 180,E1 -12602.181,E2 -12602.181} C_VEL
LIN {X 0,Y 369.202,Z 262.113,A -85,B 0,C 180,E1 -12606.558,E2 -12606.558} C_VEL
LIN {X 0,Y 369.131,Z 262.128,A -85,B 0,C 180,E1 -12608.761,E2 -12608.761} C_VEL
LIN {X 0,Y 368.998,Z 262.139,A -85,B 0,C 180,E1 -12612.093,E2 -12612.093} C_VEL
LIN {X 0,Y 368.991,Z 262.14,A -85,B 0,C 180,E1 -12615.465,E2 -12615.465} C_VEL
LIN {X 0,Y 368.96,Z 262.148,A -85,B 0,C 180,E1 -12618.894,E2 -12618.894} C_VEL
LIN {X 0,Y 368.926,Z 262.156,A -85,B 0,C 180,E1 -12622.395,E2 -12622.395} C_VEL
LIN {X 0,Y 368.994,Z 262.145,A -85,B 0,C 180,E1 -12625.98,E2 -12625.98} C_VEL
LIN {X 0,Y 368.962,Z 262.139,A -85,B 0,C 180,E1 -12628.814,E2 -12628.814} C_VEL
LIN {X 0,Y 368.894,Z 262.15,A -85,B 0,C 180,E1 -12632.238,E2 -12632.238} C_VEL
LIN {X 0,Y 368.924,Z 262.152,A -85,B 0,C 180,E1 -12635.002,E2 -12635.002} C_VEL
LIN {X 0,Y 368.906,Z 262.157,A -85,B 0,C 180,E1 -12638.641,E2 -12638.641} C_VEL
LIN {X 0,Y 368.876,Z 262.148,A -85,B 0,C 180,E1 -12642.01,E2 -12642.01} C_VEL
LIN {X 0,Y 368.922,Z 262.153,A -85,B 0,C 180,E1 -12645.183,E2 -12645.183} C_VEL
LIN {X 0,Y 368.878,Z 262.116,A -85,B 0,C 180,E1 -12648.178,E2 -12648.178} C_VEL
LIN {X 0,Y 368.907,Z 262.16,A -85,B 0,C 180,E1 -12651.36,E2 -12651.36} C_VEL
LIN {X 0,Y 368.934,Z 262.131,A -85,B 0,C 180,E1 -12655.147,E2 -12655.147} C_VEL
LIN {X 0,Y 368.934,Z 262.378,A -85,B 0,C 180,E1 -12657.199,E2 -12657.199} C_VEL
LIN {X 0,Y 372.402,Z 275.614,A -85,B 0,C 180,E1 -12660.24,E2 -12660.24} C_VEL
LIN {X 0,Y 375.381,Z 288.405,A -85,B 0,C 180,E1 -12662.999,E2 -12662.999} C_VEL
LIN {X 0,Y 375.922,Z 291.818,A -85,B 0,C 180,E1 -12663.699,E2 -12663.699} C_VEL
LIN {X 0,Y 375.153,Z 298.893,A -85,B 0,C 180,E1 -12664.956,E2 -12664.956} C_VEL
LIN {X 0,Y 379.088,Z 325.478,A -85,B 0,C 180,E1 -12665.784,E2 -12665.784} C_VEL
LIN {X 0,Y 376.96,Z 430.636,A -85,B 0,C 180,E1 -12667.891,E2 -12667.891} C_VEL
LIN {X 0,Y 376.27,Z 444.581,A -85,B 0,C 180,E1 -12668.353,E2 -12668.353} C_VEL
LIN {X 0,Y 375.457,Z 458.166,A -85,B 0,C 180,E1 -12669.024,E2 -12669.024} C_VEL
LIN {X 0,Y 374.523,Z 470.714,A -85,B 0,C 180,E1 -12669.848,E2 -12669.848} C_VEL
LIN {X 0,Y 373.387,Z 483.398,A -85,B 0,C 180,E1 -12670.911,E2 -12670.911} C_VEL
LIN {X 0,Y 372.147,Z 495.1,A -85,B 0,C 180,E1 -12672.129,E2 -12672.129} C_VEL
LIN {X 0,Y 371.023,Z 505.798,A -85,B 0,C 180,E1 -12673.493,E2 -12673.493} C_VEL
LIN {X 0,Y 369.992,Z 516.391,A -85,B 0,C 180,E1 -12675.142,E2 -12675.142} C_VEL
LIN {X 0,Y 369.214,Z 525.083,A -85,B 0,C 180,E1 -12676.796,E2 -12676.796} C_VEL
LIN {X 0,Y 368.387,Z 533.328,A -85,B 0,C 180,E1 -12678.724,E2 -12678.724} C_VEL
LIN {X 0,Y 367.871,Z 539.939,A -85,B 0,C 180,E1 -12680.655,E2 -12680.655} C_VEL
LIN {X 0,Y 367.626,Z 544.486,A -85,B 0,C 180,E1 -12682.31,E2 -12682.31} C_VEL
LIN {X 0,Y 367.449,Z 548.186,A -85,B 0,C 180,E1 -12684.028,E2 -12684.028} C_VEL
LIN {X 0,Y 367.412,Z 550.719,A -85,B 0,C 180,E1 -12685.612,E2 -12685.612} C_VEL
LIN {X 0,Y 367.357,Z 552.998,A -85,B 0,C 180,E1 -12687.807,E2 -12687.807} C_VEL
LIN {X 0,Y 367.455,Z 553.851,A -85,B 0,C 180,E1 -12690,E2 -12690} C_VEL
LIN {X 0,Y 367.356,Z 553.278,A -85,B 0,C 180,E1 -12692.193,E2 -12692.193} C_VEL
LIN {X 0,Y 367.417,Z 551.26,A -85,B 0,C 180,E1 -12694.388,E2 -12694.388} C_VEL
LIN {X 0,Y 367.55,Z 547.756,A -85,B 0,C 180,E1 -12696.588,E2 -12696.588} C_VEL
LIN {X 0,Y 367.808,Z 542.682,A -85,B 0,C 180,E1 -12698.793,E2 -12698.793} C_VEL
LIN {X 0,Y 368.183,Z 537.753,A -85,B 0,C 180,E1 -12700.448,E2 -12700.448} C_VEL
LIN {X 0,Y 368.938,Z 530.609,A -85,B 0,C 180,E1 -12702.375,E2 -12702.375} C_VEL
LIN {X 0,Y 369.833,Z 521.904,A -85,B 0,C 180,E1 -12704.266,E2 -12704.266} C_VEL
LIN {X 0,Y 370.861,Z 512.406,A -85,B 0,C 180,E1 -12705.949,E2 -12705.949} C_VEL
LIN {X 0,Y 372.078,Z 502.063,A -85,B 0,C 180,E1 -12707.449,E2 -12707.449} C_VEL
LIN {X 0,Y 373.369,Z 490.601,A -85,B 0,C 180,E1 -12708.805,E2 -12708.805} C_VEL
LIN {X 0,Y 374.633,Z 479.243,A -85,B 0,C 180,E1 -12709.898,E2 -12709.898} C_VEL
LIN {X 0,Y 375.68,Z 467.464,A -85,B 0,C 180,E1 -12710.82,E2 -12710.82} C_VEL
LIN {X 0,Y 376.699,Z 454.28,A -85,B 0,C 180,E1 -12711.621,E2 -12711.621} C_VEL
LIN {X 0,Y 377.589,Z 439.979,A -85,B 0,C 180,E1 -12712.25,E2 -12712.25} C_VEL
LIN {X 0,Y 378.177,Z 426.055,A -85,B 0,C 180,E1 -12712.646,E2 -12712.646} C_VEL
LIN {X 0,Y 380.268,Z 325.263,A -85,B 0,C 180,E1 -12714.66,E2 -12714.66} C_VEL
LIN {X 0,Y 375.975,Z 298.926,A -85,B 0,C 180,E1 -12715.543,E2 -12715.543} C_VEL
LIN {X 0,Y 376.573,Z 293.009,A -85,B 0,C 180,E1 -12716.609,E2 -12716.609} C_VEL
LIN {X 0,Y 374.554,Z 283.704,A -85,B 0,C 180,E1 -12718.616,E2 -12718.616} C_VEL
LIN {X 0,Y 371.247,Z 270.683,A -85,B 0,C 180,E1 -12721.583,E2 -12721.583} C_VEL
LIN {X 0,Y 368.96,Z 262.246,A -85,B 0,C 180,E1 -12723.654,E2 -12723.654} C_VEL
LIN {X 0,Y 368.901,Z 262.133,A -85,B 0,C 180,E1 -12727.563,E2 -12727.563} C_VEL
LIN {X 0,Y 368.95,Z 262.144,A -85,B 0,C 180,E1 -12730.364,E2 -12730.364} C_VEL
LIN {X 0,Y 368.955,Z 262.145,A -85,B 0,C 180,E1 -12733.628,E2 -12733.628} C_VEL
LIN {X 0,Y 368.886,Z 262.16,A -85,B 0,C 180,E1 -12736.696,E2 -12736.696} C_VEL
LIN {X 0,Y 368.908,Z 262.146,A -85,B 0,C 180,E1 -12739.643,E2 -12739.643} C_VEL
LIN {X 0,Y 368.898,Z 262.144,A -85,B 0,C 180,E1 -12743.144,E2 -12743.144} C_VEL
LIN {X 0,Y 368.892,Z 262.161,A -85,B 0,C 180,E1 -12746.462,E2 -12746.462} C_VEL
LIN {X 0,Y 368.918,Z 262.131,A -85,B 0,C 180,E1 -12750.31,E2 -12750.31} C_VEL
LIN {X 0,Y 368.976,Z 262.148,A -85,B 0,C 180,E1 -12753.535,E2 -12753.535} C_VEL
LIN {X 0,Y 368.961,Z 262.15,A -85,B 0,C 180,E1 -12756.421,E2 -12756.421} C_VEL
LIN {X 0,Y 368.931,Z 262.149,A -85,B 0,C 180,E1 -12759.947,E2 -12759.947} C_VEL
LIN {X 0,Y 368.97,Z 262.143,A -85,B 0,C 180,E1 -12763.399,E2 -12763.399} C_VEL
LIN {X 0,Y 369.052,Z 262.135,A -85,B 0,C 180,E1 -12766.79,E2 -12766.79} C_VEL
LIN {X 0,Y 369.061,Z 262.138,A -85,B 0,C 180,E1 -12770.132,E2 -12770.132} C_VEL
LIN {X 0,Y 369.157,Z 262.115,A -85,B 0,C 180,E1 -12772.342,E2 -12772.342} C_VEL
LIN {X 0,Y 369.138,Z 262.126,A -85,B 0,C 180,E1 -12774.538,E2 -12774.538} C_VEL
LIN {X 0,Y 369.313,Z 262.099,A -85,B 0,C 180,E1 -12777.819,E2 -12777.819} C_VEL
LIN {X 0,Y 369.452,Z 262.089,A -85,B 0,C 180,E1 -12780,E2 -12780} C_VEL
LIN {X 0,Y 369.313,Z 262.096,A -85,B 0,C 180,E1 -12782.182,E2 -12782.182} C_VEL
LIN {X 0,Y 369.198,Z 262.113,A -85,B 0,C 180,E1 -12786.621,E2 -12786.621} C_VEL
LIN {X 0,Y 369.133,Z 262.126,A -85,B 0,C 180,E1 -12788.761,E2 -12788.761} C_VEL
LIN {X 0,Y 369,Z 262.14,A -85,B 0,C 180,E1 -12792.094,E2 -12792.094} C_VEL
LIN {X 0,Y 368.993,Z 262.14,A -85,B 0,C 180,E1 -12795.465,E2 -12795.465} C_VEL
LIN {X 0,Y 368.954,Z 262.152,A -85,B 0,C 180,E1 -12798.895,E2 -12798.895} C_VEL
LIN {X 0,Y 368.932,Z 262.153,A -85,B 0,C 180,E1 -12802.396,E2 -12802.396} C_VEL
LIN {X 0,Y 368.997,Z 262.145,A -85,B 0,C 180,E1 -12805.981,E2 -12805.981} C_VEL
LIN {X 0,Y 368.912,Z 262.137,A -85,B 0,C 180,E1 -12809.691,E2 -12809.691} C_VEL
LIN {X 0,Y 368.895,Z 262.156,A -85,B 0,C 180,E1 -12813.044,E2 -12813.044} C_VEL
LIN {X 0,Y 368.916,Z 262.147,A -85,B 0,C 180,E1 -12816.198,E2 -12816.198} C_VEL
LIN {X 0,Y 368.902,Z 262.148,A -85,B 0,C 180,E1 -12818.954,E2 -12818.954} C_VEL
LIN {X 0,Y 368.881,Z 262.16,A -85,B 0,C 180,E1 -12822.01,E2 -12822.01} C_VEL
LIN {X 0,Y 368.881,Z 262.157,A -85,B 0,C 180,E1 -12825.177,E2 -12825.177} C_VEL
LIN {X 0,Y 368.884,Z 262.153,A -85,B 0,C 180,E1 -12828.179,E2 -12828.179} C_VEL
LIN {X 0,Y 368.909,Z 262.125,A -85,B 0,C 180,E1 -12831.361,E2 -12831.361} C_VEL
LIN {X 0,Y 368.977,Z 262.316,A -85,B 0,C 180,E1 -12833.993,E2 -12833.993} C_VEL
LIN {X 0,Y 371.723,Z 272.953,A -85,B 0,C 180,E1 -12836.751,E2 -12836.751} C_VEL
LIN {X 0,Y 374.743,Z 285.958,A -85,B 0,C 180,E1 -12839.918,E2 -12839.918} C_VEL
LIN {X 0,Y 375.658,Z 291.195,A -85,B 0,C 180,E1 -12841.129,E2 -12841.129} C_VEL
LIN {X 0,Y 373.894,Z 307.478,A -85,B 0,C 180,E1 -12844.456,E2 -12844.456} C_VEL
LIN {X 0,Y 373.476,Z 312.231,A -85,B 0,C 180,E1 -12845.347,E2 -12845.347} C_VEL
LIN {X 0,Y 379.363,Z 343.528,A -85,B 0,C 180,E1 -12846.378,E2 -12846.378} C_VEL
LIN {X 0,Y 378.499,Z 402.958,A -85,B 0,C 180,E1 -12847.447,E2 -12847.447} C_VEL
LIN {X 0,Y 378.064,Z 427.541,A -85,B 0,C 180,E1 -12847.923,E2 -12847.923} C_VEL
LIN {X 0,Y 377.409,Z 440.616,A -85,B 0,C 180,E1 -12848.378,E2 -12848.378} C_VEL
LIN {X 0,Y 376.66,Z 453.563,A -85,B 0,C 180,E1 -12849.062,E2 -12849.062} C_VEL
LIN {X 0,Y 375.618,Z 465.23,A -85,B 0,C 180,E1 -12849.891,E2 -12849.891} C_VEL
LIN {X 0,Y 374.373,Z 476.835,A -85,B 0,C 180,E1 -12850.963,E2 -12850.963} C_VEL
LIN {X 0,Y 373.088,Z 487.279,A -85,B 0,C 180,E1 -12852.175,E2 -12852.175} C_VEL
LIN {X 0,Y 371.84,Z 496.72,A -85,B 0,C 180,E1 -12853.531,E2 -12853.531} C_VEL
LIN {X 0,Y 370.711,Z 504.999,A -85,B 0,C 180,E1 -12854.991,E2 -12854.991} C_VEL
LIN {X 0,Y 369.889,Z 512.125,A -85,B 0,C 180,E1 -12856.541,E2 -12856.541} C_VEL
LIN {X 0,Y 369.129,Z 517.334,A -85,B 0,C 180,E1 -12857.911,E2 -12857.911} C_VEL
LIN {X 0,Y 368.46,Z 522.451,A -85,B 0,C 180,E1 -12859.56,E2 -12859.56} C_VEL
LIN {X 0,Y 368.042,Z 526.46,A -85,B 0,C 180,E1 -12861.213,E2 -12861.213} C_VEL
LIN {X 0,Y 367.843,Z 528.6,A -85,B 0,C 180,E1 -12862.314,E2 -12862.314} C_VEL
LIN {X 0,Y 367.534,Z 531.588,A -85,B 0,C 180,E1 -12864.514,E2 -12864.514} C_VEL
LIN {X 0,Y 367.502,Z 532.512,A -85,B 0,C 180,E1 -12865.613,E2 -12865.613} C_VEL
LIN {X 0,Y 367.413,Z 533.281,A -85,B 0,C 180,E1 -12867.808,E2 -12867.808} C_VEL
LIN {X 0,Y 367.461,Z 532.542,A -85,B 0,C 180,E1 -12870,E2 -12870} C_VEL
LIN {X 0,Y 367.615,Z 530.348,A -85,B 0,C 180,E1 -12872.191,E2 -12872.191} C_VEL
LIN {X 0,Y 367.896,Z 527.665,A -85,B 0,C 180,E1 -12873.834,E2 -12873.834} C_VEL
LIN {X 0,Y 368.129,Z 524.044,A -85,B 0,C 180,E1 -12875.477,E2 -12875.477} C_VEL
LIN {X 0,Y 368.702,Z 518.825,A -85,B 0,C 180,E1 -12877.288,E2 -12877.288} C_VEL
LIN {X 0,Y 369.39,Z 512.427,A -85,B 0,C 180,E1 -12879.031,E2 -12879.031} C_VEL
LIN {X 0,Y 370.313,Z 504.925,A -85,B 0,C 180,E1 -12880.663,E2 -12880.663} C_VEL
LIN {X 0,Y 371.437,Z 495.559,A -85,B 0,C 180,E1 -12882.29,E2 -12882.29} C_VEL
LIN {X 0,Y 372.485,Z 485.948,A -85,B 0,C 180,E1 -12883.641,E2 -12883.641} C_VEL
LIN {X 0,Y 373.705,Z 475.28,A -85,B 0,C 180,E1 -12884.846,E2 -12884.846} C_VEL
LIN {X 0,Y 374.072,Z 470.432,A -85,B 0,C 180,E1 -12885.315,E2 -12885.315} C_VEL
LIN {X 0,Y 374.019,Z 465.381,A -85,B 0,C 180,E1 -12885.787,E2 -12885.787} C_VEL
LIN {X 0,Y 371.984,Z 457.04,A -85,B 0,C 180,E1 -12886.557,E2 -12886.557} C_VEL
LIN {X 0,Y 369.854,Z 448.383,A -85,B 0,C 180,E1 -12887.23,E2 -12887.23} C_VEL
LIN {X 0,Y 369.639,Z 442.84,A -85,B 0,C 180,E1 -12887.543,E2 -12887.543} C_VEL
LIN {X 0,Y 370.194,Z 430.942,A -85,B 0,C 180,E1 -12888.011,E2 -12888.011} C_VEL
LIN {X 0,Y 370.551,Z 415.328,A -85,B 0,C 180,E1 -12888.368,E2 -12888.368} C_VEL
LIN {X 0,Y 371.547,Z 344.056,A -85,B 0,C 180,E1 -12889.668,E2 -12889.668} C_VEL
LIN {X 0,Y 366.303,Z 313.715,A -85,B 0,C 180,E1 -12890.598,E2 -12890.598} C_VEL
LIN {X 0,Y 366.043,Z 311.569,A -85,B 0,C 180,E1 -12890.732,E2 -12890.732} C_VEL
LIN {X 0,Y 367.793,Z 294.334,A -85,B 0,C 180,E1 -12894.257,E2 -12894.257} C_VEL
LIN {X 0,Y 368.116,Z 290.291,A -85,B 0,C 180,E1 -12895.107,E2 -12895.107} C_VEL
LIN {X 0,Y 365.428,Z 277.253,A -85,B 0,C 180,E1 -12898.204,E2 -12898.204} C_VEL
LIN {X 0,Y 362.258,Z 264.612,A -85,B 0,C 180,E1 -12901.391,E2 -12901.391} C_VEL
LIN {X 0,Y 361.88,Z 263.074,A -85,B 0,C 180,E1 -12901.87,E2 -12901.87} C_VEL
LIN {X 0,Y 361.869,Z 263.03,A -85,B 0,C 180,E1 -12905.636,E2 -12905.636} C_VEL
LIN {X 0,Y 361.87,Z 263.034,A -85,B 0,C 180,E1 -12909.026,E2 -12909.026} C_VEL
LIN {X 0,Y 361.837,Z 263.038,A -85,B 0,C 180,E1 -12912.828,E2 -12912.828} C_VEL
LIN {X 0,Y 361.817,Z 263.031,A -85,B 0,C 180,E1 -12915.946,E2 -12915.946} C_VEL
LIN {X 0,Y 361.833,Z 263.023,A -85,B 0,C 180,E1 -12919.244,E2 -12919.244} C_VEL
LIN {X 0,Y 361.862,Z 263.035,A -85,B 0,C 180,E1 -12922.776,E2 -12922.776} C_VEL
LIN {X 0,Y 361.852,Z 263.013,A -85,B 0,C 180,E1 -12925.719,E2 -12925.719} C_VEL
LIN {X 0,Y 361.873,Z 263.033,A -85,B 0,C 180,E1 -12929.671,E2 -12929.671} C_VEL
LIN {X 0,Y 361.951,Z 263.023,A -85,B 0,C 180,E1 -12933.474,E2 -12933.474} C_VEL
LIN {X 0,Y 361.88,Z 263.033,A -85,B 0,C 180,E1 -12937.143,E2 -12937.143} C_VEL
LIN {X 0,Y 361.902,Z 263.023,A -85,B 0,C 180,E1 -12940.723,E2 -12940.723} C_VEL
LIN {X 0,Y 361.928,Z 263.026,A -85,B 0,C 180,E1 -12943.065,E2 -12943.065} C_VEL
LIN {X 0,Y 361.993,Z 263.015,A -85,B 0,C 180,E1 -12946.527,E2 -12946.527} C_VEL
LIN {X 0,Y 362.026,Z 263.005,A -85,B 0,C 180,E1 -12949.937,E2 -12949.937} C_VEL
LIN {X 0,Y 362.157,Z 262.995,A -85,B 0,C 180,E1 -12953.313,E2 -12953.313} C_VEL
LIN {X 0,Y 362.277,Z 262.981,A -85,B 0,C 180,E1 -12957.776,E2 -12957.776} C_VEL
LIN {X 0,Y 362.421,Z 262.959,A -85,B 0,C 180,E1 -12960,E2 -12960} C_VEL
LIN {X 0,Y 362.276,Z 262.979,A -85,B 0,C 180,E1 -12962.223,E2 -12962.223} C_VEL
LIN {X 0,Y 362.165,Z 262.99,A -85,B 0,C 180,E1 -12966.686,E2 -12966.686} C_VEL
LIN {X 0,Y 362.068,Z 263.007,A -85,B 0,C 180,E1 -12968.933,E2 -12968.933} C_VEL
LIN {X 0,Y 361.953,Z 263.02,A -85,B 0,C 180,E1 -12972.332,E2 -12972.332} C_VEL
LIN {X 0,Y 361.956,Z 263.019,A -85,B 0,C 180,E1 -12974.62,E2 -12974.62} C_VEL
LIN {X 0,Y 361.951,Z 263.025,A -85,B 0,C 180,E1 -12978.099,E2 -12978.099} C_VEL
LIN {X 0,Y 361.886,Z 263.027,A -85,B 0,C 180,E1 -12981.653,E2 -12981.653} C_VEL
LIN {X 0,Y 361.922,Z 263.02,A -85,B 0,C 180,E1 -12985.29,E2 -12985.29} C_VEL
LIN {X 0,Y 361.917,Z 263.026,A -85,B 0,C 180,E1 -12987.778,E2 -12987.778} C_VEL
LIN {X 0,Y 361.841,Z 263.017,A -85,B 0,C 180,E1 -12991.286,E2 -12991.286} C_VEL
